(* IEC 61131-3 sources: SmartHomeNew/ (part 12) *)

(* ---- PRG_Epistemic_Integrity_Governor.st ---- *)
PROGRAM PRG_Epistemic_Integrity_Governor
VAR
    L_Now_MS : UDINT;
    L_Epistemic_Valid : BOOL := TRUE;
    L_Error_Code : UDINT := 0;
    L_Error_Text : STRING(160) := '';
END_VAR

L_Now_MS := GVL_STATUS.G_System_Time_MS;
L_Epistemic_Valid := TRUE;
L_Error_Code := 0;
L_Error_Text := '';

// Fail-safe defaults.
GVL_EPISTEMIC_INTEGRITY_FABRIC.Epistemic_Integrity_Valid := FALSE;
GVL_EPISTEMIC_INTEGRITY_FABRIC.Epistemic_Integrity_Granted := FALSE;
GVL_EPISTEMIC_INTEGRITY_FABRIC.Epistemic_Integrity_Quarantine_Active := TRUE;

GVL_EPISTEMIC_INTEGRITY_FABRIC.Physical_Reality_Model_Coherent := FALSE;
GVL_EPISTEMIC_INTEGRITY_FABRIC.Sensor_Truth_Consensus_Valid := FALSE;
GVL_EPISTEMIC_INTEGRITY_FABRIC.Telemetry_Reality_Alignment_Stable := FALSE;
GVL_EPISTEMIC_INTEGRITY_FABRIC.Distributed_Reality_Model_Consistent := FALSE;
GVL_EPISTEMIC_INTEGRITY_FABRIC.Causal_Model_Physically_Valid := FALSE;

// Forensic evidence required.
IF NOT GVL_FORENSIC_EVIDENCE_FABRIC.Forensic_Evidence_Granted THEN
    L_Epistemic_Valid := FALSE;
    L_Error_Code := 44000;
    L_Error_Text := 'Forensic evidence authority not granted';
END_IF;

// Epistemic split-brain detectors.
IF GVL_EPISTEMIC_INTEGRITY_FABRIC.Physically_False_Consensus_Detected THEN
    L_Epistemic_Valid := FALSE;
    L_Error_Code := 44001;
    L_Error_Text := 'Physically false consensus detected';
END_IF;

IF GVL_EPISTEMIC_INTEGRITY_FABRIC.Telemetry_Corruption_Coherent_Detected THEN
    L_Epistemic_Valid := FALSE;
    L_Error_Code := 44002;
    L_Error_Text := 'Telemetry corruption coherence detected';
END_IF;

IF GVL_EPISTEMIC_INTEGRITY_FABRIC.Historical_Reality_Divergence_Detected THEN
    L_Epistemic_Valid := FALSE;
    L_Error_Code := 44003;
    L_Error_Text := 'Historical reality divergence detected';
END_IF;

IF GVL_EPISTEMIC_INTEGRITY_FABRIC.Sensor_Trust_Erosion_Detected THEN
    L_Epistemic_Valid := FALSE;
    L_Error_Code := 44004;
    L_Error_Text := 'Sensor trust erosion detected';
END_IF;

IF GVL_EPISTEMIC_INTEGRITY_FABRIC.Causal_Model_Poisoning_Detected THEN
    L_Epistemic_Valid := FALSE;
    L_Error_Code := 44005;
    L_Error_Text := 'Causal model poisoning detected';
END_IF;

IF GVL_EPISTEMIC_INTEGRITY_FABRIC.LongTerm_Epistemic_Drift_Detected THEN
    L_Epistemic_Valid := FALSE;
    L_Error_Code := 44006;
    L_Error_Text := 'Long-term epistemic drift detected';
END_IF;

// Physical reality anchoring validation.
IF L_Epistemic_Valid
AND NOT GVL_EPISTEMIC_INTEGRITY_FABRIC.Historical_Reality_Anchoring_Valid THEN
    L_Epistemic_Valid := FALSE;
    L_Error_Code := 44010;
    L_Error_Text := 'Historical reality anchoring invalid';
END_IF;

IF L_Epistemic_Valid
AND NOT GVL_EPISTEMIC_INTEGRITY_FABRIC.Physical_Truth_Lineage_Coherent THEN
    L_Epistemic_Valid := FALSE;
    L_Error_Code := 44011;
    L_Error_Text := 'Physical truth lineage coherence invalid';
END_IF;

IF L_Epistemic_Valid
AND NOT GVL_EPISTEMIC_INTEGRITY_FABRIC.Reality_Model_Drift_Bounded THEN
    L_Epistemic_Valid := FALSE;
    L_Error_Code := 44012;
    L_Error_Text := 'Reality model drift bounds invalid';
END_IF;

IF L_Epistemic_Valid
AND NOT GVL_EPISTEMIC_INTEGRITY_FABRIC.Semantic_To_Physical_Causality_Valid THEN
    L_Epistemic_Valid := FALSE;
    L_Error_Code := 44013;
    L_Error_Text := 'Semantic-to-physical causality invalid';
END_IF;

IF L_Epistemic_Valid THEN
    GVL_EPISTEMIC_INTEGRITY_FABRIC.Epistemic_Integrity_Valid := TRUE;
    GVL_EPISTEMIC_INTEGRITY_FABRIC.Epistemic_Integrity_Granted := TRUE;
    GVL_EPISTEMIC_INTEGRITY_FABRIC.Epistemic_Integrity_Quarantine_Active := FALSE;

    GVL_EPISTEMIC_INTEGRITY_FABRIC.Physical_Reality_Model_Coherent := TRUE;
    GVL_EPISTEMIC_INTEGRITY_FABRIC.Sensor_Truth_Consensus_Valid := TRUE;
    GVL_EPISTEMIC_INTEGRITY_FABRIC.Telemetry_Reality_Alignment_Stable := TRUE;
    GVL_EPISTEMIC_INTEGRITY_FABRIC.Distributed_Reality_Model_Consistent := TRUE;
    GVL_EPISTEMIC_INTEGRITY_FABRIC.Causal_Model_Physically_Valid := TRUE;

    GVL_EPISTEMIC_INTEGRITY_FABRIC.Epistemic_Integrity_Epoch :=
        GVL_FORENSIC_EVIDENCE_FABRIC.Forensic_Evidence_Epoch;

    GVL_EPISTEMIC_INTEGRITY_FABRIC.Epistemic_Integrity_Epoch_Coherent := TRUE;

    GVL_EPISTEMIC_INTEGRITY_FABRIC.Epistemic_Integrity_Last_Update_MS :=
        L_Now_MS;

    GVL_EPISTEMIC_INTEGRITY_FABRIC.Epistemic_Integrity_Lease_Expired := FALSE;

    GVL_EPISTEMIC_INTEGRITY_FABRIC.Epistemic_Integrity_Last_Error_Code := 0;
    GVL_EPISTEMIC_INTEGRITY_FABRIC.Epistemic_Integrity_Last_Error_Text := '';
ELSE
    GVL_EPISTEMIC_INTEGRITY_FABRIC.Epistemic_Integrity_Valid := FALSE;
    GVL_EPISTEMIC_INTEGRITY_FABRIC.Epistemic_Integrity_Granted := FALSE;
    GVL_EPISTEMIC_INTEGRITY_FABRIC.Epistemic_Integrity_Quarantine_Active := TRUE;

    GVL_EPISTEMIC_INTEGRITY_FABRIC.Epistemic_Integrity_Lease_Expired := TRUE;

    GVL_EPISTEMIC_INTEGRITY_FABRIC.Epistemic_Integrity_Last_Error_Code :=
        L_Error_Code;

    GVL_EPISTEMIC_INTEGRITY_FABRIC.Epistemic_Integrity_Last_Error_Text :=
        L_Error_Text;

    GVL_EPISTEMIC_INTEGRITY_FABRIC.Epistemic_Integrity_Invalidation_Count :=
        GVL_EPISTEMIC_INTEGRITY_FABRIC.Epistemic_Integrity_Invalidation_Count + 1;
END_IF;

END_PROGRAM

(* ---- PRG_Execution_Progress_Causality_Governor.st ---- *)
PROGRAM PRG_Execution_Progress_Causality_Governor
IF GVL_PHYSICAL_DEADLOCK_RESOLUTION_FABRIC.Physical_Deadlock_Resolution_Granted
AND NOT GVL_EXECUTION_PROGRESS_CAUSALITY_FABRIC.Distributed_Execution_Stall_Detected
AND NOT GVL_EXECUTION_PROGRESS_CAUSALITY_FABRIC.Execution_Progress_Divergence_Detected
AND NOT GVL_EXECUTION_PROGRESS_CAUSALITY_FABRIC.Recovery_Progress_Oscillation_Detected THEN

    GVL_EXECUTION_PROGRESS_CAUSALITY_FABRIC.Execution_Progress_Causality_Valid := TRUE;
    GVL_EXECUTION_PROGRESS_CAUSALITY_FABRIC.Execution_Progress_Causality_Granted := TRUE;
    GVL_EXECUTION_PROGRESS_CAUSALITY_FABRIC.Progress_Causality_Grounded := TRUE;
    GVL_EXECUTION_PROGRESS_CAUSALITY_FABRIC.Deterministic_Execution_Continuation_Valid := TRUE;
END_IF;
END_PROGRAM

(* ---- PRG_Explainability.st ---- *)
PROGRAM PRG_Explainability
VAR
    L_Mode : E_Safety_Mode;
    L_Recovery : E_Recovery_Phase;
END_VAR

L_Mode := GVL_SAFETY_SHUTDOWN.G_Safety_Mode;
L_Recovery := GVL_SAFETY_RECOVERY.G_Recovery_Phase;

GVL_EXPLAINABILITY.G_Last_Safety_Mode := L_Mode;
GVL_EXPLAINABILITY.G_Last_Recovery_Phase := L_Recovery;
GVL_EXPLAINABILITY.G_Last_Update_MS := GVL_TIME_SERVICE.G_Now_MS;

// Global reason
CASE L_Mode OF
    FIRE:
        GVL_EXPLAINABILITY.G_Last_Global_Reason_Code := REASON_FIRE;
        GVL_EXPLAINABILITY.G_Last_Global_Reason_Text := 'Fire safety mode active';
    GAS:
        GVL_EXPLAINABILITY.G_Last_Global_Reason_Code := REASON_GAS;
        GVL_EXPLAINABILITY.G_Last_Global_Reason_Text := 'Gas safety mode active';
    WATER_LEAK:
        GVL_EXPLAINABILITY.G_Last_Global_Reason_Code := REASON_WATER_LEAK;
        GVL_EXPLAINABILITY.G_Last_Global_Reason_Text := 'Water leak detected';
    GLOBAL_STOP:
        GVL_EXPLAINABILITY.G_Last_Global_Reason_Code := REASON_GLOBAL_STOP;
        GVL_EXPLAINABILITY.G_Last_Global_Reason_Text := 'Global stop active';
    EVACUATION:
        GVL_EXPLAINABILITY.G_Last_Global_Reason_Code := REASON_EVACUATION;
        GVL_EXPLAINABILITY.G_Last_Global_Reason_Text := 'Evacuation mode active';
    NORMAL:
        IF GVL_SAFETY_RECOVERY.G_Recovery_Active THEN
            GVL_EXPLAINABILITY.G_Last_Global_Reason_Code := REASON_RECOVERY_ACTIVE;
            GVL_EXPLAINABILITY.G_Last_Global_Reason_Text := 'System in recovery phase';
        ELSE
            GVL_EXPLAINABILITY.G_Last_Global_Reason_Code := REASON_NONE;
            GVL_EXPLAINABILITY.G_Last_Global_Reason_Text := 'System in normal operation';
        END_IF;
END_CASE;

// Domain explanations
IF GVL_COMMAND_SHADOW.G_Heating_Block THEN
    GVL_EXPLAINABILITY.G_Heating_Why_Blocked := 'Heating blocked by command arbitration (safety or recovery)';
ELSE
    GVL_EXPLAINABILITY.G_Heating_Why_Blocked := '';
END_IF;

IF GVL_COMMAND_SHADOW.G_Vent_Stop THEN
    GVL_EXPLAINABILITY.G_Vent_Why_Stopped := 'Ventilation stopped by command arbitration';
ELSE
    GVL_EXPLAINABILITY.G_Vent_Why_Stopped := '';
END_IF;

IF GVL_COMMAND_SHADOW.G_Close_Valve_35 OR GVL_COMMAND_SHADOW.G_Close_Valve_36 THEN
    GVL_EXPLAINABILITY.G_Water_Why_Closed := 'Water valves closed by safety command';
ELSE
    GVL_EXPLAINABILITY.G_Water_Why_Closed := '';
END_IF;

IF GVL_COMMAND_SHADOW.G_Lock_1_Open OR GVL_COMMAND_SHADOW.G_Lock_2_Open THEN
    GVL_EXPLAINABILITY.G_Access_Why_Opened := 'Access opened due to evacuation or command override';
ELSE
    GVL_EXPLAINABILITY.G_Access_Why_Opened := '';
END_IF;

// >>> BULK_SYNC_ANCHOR: PRG_Explainability <<<

(* ---- PRG_File_Archive_HMI_Applicator.st ---- *)
PROGRAM PRG_File_Archive_HMI_Applicator
// ==============================================================================
// FILE ARCHIVE HMI APPLICATOR — validates HMI intent and updates archive runtime.
// ==============================================================================
// HMI is not allowed to write files or physical outputs directly. This program
// only transfers validated one-shot requests/configuration into GVL_FILE_ARCHIVE,
// where PRG_File_Archive_Manager consumes them and publishes deterministic status.
// ==============================================================================
VAR
    L_Any_Write_Request : BOOL;
END_VAR

L_Any_Write_Request :=
    GVL_FILE_ARCHIVE_HMI.G_Write_Event_CSV_Req
    OR GVL_FILE_ARCHIVE_HMI.G_Write_Trend_CSV_Req
    OR GVL_FILE_ARCHIVE_HMI.G_Write_BlackBox_CSV_Req
    OR GVL_FILE_ARCHIVE_HMI.G_Write_Config_Backup_Req;

IF GVL_FILE_ARCHIVE_HMI.G_Set_Archive_Config_Req THEN
    IF GVL_FILE_ARCHIVE_HMI.G_File_Archive_Target_Code <= 3 THEN
        GVL_FILE_ARCHIVE.G_Archive_Interface_Enabled := GVL_FILE_ARCHIVE_HMI.G_Archive_Interface_Enabled;
        GVL_FILE_ARCHIVE.G_CSV_Write_Enabled := GVL_FILE_ARCHIVE_HMI.G_CSV_Write_Enabled;
        GVL_FILE_ARCHIVE.G_File_Archive_Target_Code := GVL_FILE_ARCHIVE_HMI.G_File_Archive_Target_Code;

        GVL_FILE_ARCHIVE_HMI.G_Last_Error := FALSE;
        GVL_FILE_ARCHIVE_HMI.G_Last_Error_Code := 0;
        GVL_FILE_ARCHIVE_HMI.G_Last_Status_Text := 'Archive configuration applied';
    ELSE
        GVL_FILE_ARCHIVE_HMI.G_Last_Error := TRUE;
        GVL_FILE_ARCHIVE_HMI.G_Last_Error_Code := 16#A101;
        GVL_FILE_ARCHIVE_HMI.G_Last_Status_Text := 'Archive configuration rejected: invalid target';
    END_IF;

    GVL_FILE_ARCHIVE_HMI.G_Last_Update_MS := GVL_TIME_SERVICE.G_Now_MS;
    GVL_FILE_ARCHIVE_HMI.G_Set_Archive_Config_Req := FALSE;
END_IF;

IF L_Any_Write_Request THEN
    IF NOT GVL_FILE_ARCHIVE.G_Archive_Interface_Enabled THEN
        GVL_FILE_ARCHIVE_HMI.G_Last_Error := TRUE;
        GVL_FILE_ARCHIVE_HMI.G_Last_Error_Code := 16#A102;
        GVL_FILE_ARCHIVE_HMI.G_Last_Status_Text := 'Archive write rejected: interface disabled';
    ELSIF NOT GVL_FILE_ARCHIVE.G_CSV_Write_Enabled THEN
        GVL_FILE_ARCHIVE_HMI.G_Last_Error := TRUE;
        GVL_FILE_ARCHIVE_HMI.G_Last_Error_Code := 16#A103;
        GVL_FILE_ARCHIVE_HMI.G_Last_Status_Text := 'Archive write rejected: CSV disabled';
    ELSE
        GVL_FILE_ARCHIVE.G_Write_Event_CSV_Request :=
            GVL_FILE_ARCHIVE.G_Write_Event_CSV_Request OR GVL_FILE_ARCHIVE_HMI.G_Write_Event_CSV_Req;
        GVL_FILE_ARCHIVE.G_Write_Trend_CSV_Request :=
            GVL_FILE_ARCHIVE.G_Write_Trend_CSV_Request OR GVL_FILE_ARCHIVE_HMI.G_Write_Trend_CSV_Req;
        GVL_FILE_ARCHIVE.G_Write_BlackBox_CSV_Request :=
            GVL_FILE_ARCHIVE.G_Write_BlackBox_CSV_Request OR GVL_FILE_ARCHIVE_HMI.G_Write_BlackBox_CSV_Req;
        GVL_FILE_ARCHIVE.G_Write_Config_Backup_Request :=
            GVL_FILE_ARCHIVE.G_Write_Config_Backup_Request OR GVL_FILE_ARCHIVE_HMI.G_Write_Config_Backup_Req;

        GVL_FILE_ARCHIVE_HMI.G_Last_Error := FALSE;
        GVL_FILE_ARCHIVE_HMI.G_Last_Error_Code := 0;
        GVL_FILE_ARCHIVE_HMI.G_Last_Status_Text := 'Archive write request accepted';
    END_IF;

    GVL_FILE_ARCHIVE_HMI.G_Last_Update_MS := GVL_TIME_SERVICE.G_Now_MS;

    // HMI requests are one-shot. Runtime requests are consumed by archive manager.
    GVL_FILE_ARCHIVE_HMI.G_Write_Event_CSV_Req := FALSE;
    GVL_FILE_ARCHIVE_HMI.G_Write_Trend_CSV_Req := FALSE;
    GVL_FILE_ARCHIVE_HMI.G_Write_BlackBox_CSV_Req := FALSE;
    GVL_FILE_ARCHIVE_HMI.G_Write_Config_Backup_Req := FALSE;
END_IF;

// >>> BULK_SYNC_ANCHOR: PRG_File_Archive_HMI_Applicator <<<
END_PROGRAM

(* ---- PRG_File_Archive_Manager.st ---- *)
PROGRAM PRG_File_Archive_Manager
// ==============================================================================
// FILE ARCHIVE MANAGER — deterministic runtime surface for future CSV/file export.
// ==============================================================================
// No direct file, USB or gateway write is implemented here. This program only
// consumes one-shot archive requests, validates the configured target surface and
// publishes a deterministic status/error until concrete CODESYS file libraries
// and port-specific paths are selected.
// ==============================================================================
VAR
    L_Request_Active : BOOL;
    L_Target_Available : BOOL;
END_VAR

L_Request_Active :=
    GVL_FILE_ARCHIVE.G_Write_Event_CSV_Request
    OR GVL_FILE_ARCHIVE.G_Write_Trend_CSV_Request
    OR GVL_FILE_ARCHIVE.G_Write_BlackBox_CSV_Request
    OR GVL_FILE_ARCHIVE.G_Write_Config_Backup_Request;

L_Target_Available := FALSE;
CASE GVL_FILE_ARCHIVE.G_File_Archive_Target_Code OF
    1:
        L_Target_Available := GVL_FILE_ARCHIVE.G_PLC_File_Target_Available;
    2:
        L_Target_Available := GVL_FILE_ARCHIVE.G_USB_Target_Available;
    3:
        L_Target_Available := GVL_FILE_ARCHIVE.G_Gateway_Target_Available;
ELSE
    L_Target_Available := FALSE;
END_CASE;

IF L_Request_Active THEN
    GVL_FILE_ARCHIVE.G_Write_Busy := FALSE;
    GVL_FILE_ARCHIVE.G_Write_Done := FALSE;
    GVL_FILE_ARCHIVE.G_Write_Error := FALSE;
    GVL_FILE_ARCHIVE.G_Last_Error_Code := 0;
    GVL_FILE_ARCHIVE.G_Last_Status_Text := '';
    GVL_FILE_ARCHIVE.G_Last_Write_MS := GVL_TIME_SERVICE.G_Now_MS;

    IF NOT GVL_FILE_ARCHIVE.G_Archive_Interface_Enabled THEN
        GVL_FILE_ARCHIVE.G_Write_Error := TRUE;
        GVL_FILE_ARCHIVE.G_Last_Error_Code := 16#A001;
        GVL_FILE_ARCHIVE.G_Last_Status_Text := 'Archive interface disabled';
    ELSIF NOT GVL_FILE_ARCHIVE.G_CSV_Write_Enabled THEN
        GVL_FILE_ARCHIVE.G_Write_Error := TRUE;
        GVL_FILE_ARCHIVE.G_Last_Error_Code := 16#A002;
        GVL_FILE_ARCHIVE.G_Last_Status_Text := 'CSV archive disabled';
    ELSIF GVL_FILE_ARCHIVE.G_File_Archive_Target_Code = 0 THEN
        GVL_FILE_ARCHIVE.G_Write_Error := TRUE;
        GVL_FILE_ARCHIVE.G_Last_Error_Code := 16#A003;
        GVL_FILE_ARCHIVE.G_Last_Status_Text := 'No archive target selected';
    ELSIF NOT L_Target_Available THEN
        GVL_FILE_ARCHIVE.G_Write_Error := TRUE;
        GVL_FILE_ARCHIVE.G_Last_Error_Code := 16#A004;
        GVL_FILE_ARCHIVE.G_Last_Status_Text := 'Selected archive target unavailable';
    ELSE
        GVL_FILE_ARCHIVE.G_Write_Error := TRUE;
        GVL_FILE_ARCHIVE.G_Last_Error_Code := 16#A005;
        GVL_FILE_ARCHIVE.G_Last_Status_Text := 'Archive backend not connected';
    END_IF;

    // One-shot requests are consumed regardless of the result so HMI/gateway
    // callers receive a stable status instead of repeatedly retriggering.
    GVL_FILE_ARCHIVE.G_Write_Event_CSV_Request := FALSE;
    GVL_FILE_ARCHIVE.G_Write_Trend_CSV_Request := FALSE;
    GVL_FILE_ARCHIVE.G_Write_BlackBox_CSV_Request := FALSE;
    GVL_FILE_ARCHIVE.G_Write_Config_Backup_Request := FALSE;
END_IF;

// >>> BULK_SYNC_ANCHOR: PRG_File_Archive_Manager <<<
END_PROGRAM

(* ---- PRG_Governance_Observer_Consensus_Governor.st ---- *)
PROGRAM PRG_Governance_Observer_Consensus_Governor
VAR
    L_Now_MS : UDINT;
    L_Consensus_Valid : BOOL := TRUE;
    L_Error_Code : UDINT := 0;
    L_Error_Text : STRING(160) := '';
END_VAR

L_Now_MS := GVL_STATUS.G_System_Time_MS;
L_Consensus_Valid := TRUE;
L_Error_Code := 0;
L_Error_Text := '';

// Fail-safe defaults.
GVL_GOVERNANCE_OBSERVER_CONSENSUS_FABRIC.Governance_Observer_Consensus_Valid := FALSE;
GVL_GOVERNANCE_OBSERVER_CONSENSUS_FABRIC.Governance_Observer_Consensus_Granted := FALSE;
GVL_GOVERNANCE_OBSERVER_CONSENSUS_FABRIC.Governance_Observer_Consensus_Quarantine_Active := TRUE;

GVL_GOVERNANCE_OBSERVER_CONSENSUS_FABRIC.Distributed_Governance_Projection_Consistent := FALSE;
GVL_GOVERNANCE_OBSERVER_CONSENSUS_FABRIC.Observer_Semantic_Consensus_Valid := FALSE;
GVL_GOVERNANCE_OBSERVER_CONSENSUS_FABRIC.CrossNode_Authority_Interpretation_Aligned := FALSE;
GVL_GOVERNANCE_OBSERVER_CONSENSUS_FABRIC.Governance_Reality_Canonical := FALSE;
GVL_GOVERNANCE_OBSERVER_CONSENSUS_FABRIC.Observer_Projection_Lineage_Coherent := FALSE;

// Semantic epoch invariance required.
IF NOT GVL_SEMANTIC_EPOCH_INVARIANCE_FABRIC.Semantic_Epoch_Invariance_Granted THEN
    L_Consensus_Valid := FALSE;
    L_Error_Code := 50000;
    L_Error_Text := 'Semantic epoch invariance not granted';
END_IF;

// Governance observer split-brain detectors.
IF GVL_GOVERNANCE_OBSERVER_CONSENSUS_FABRIC.Observer_Governance_Divergence_Detected THEN
    L_Consensus_Valid := FALSE;
    L_Error_Code := 50001;
    L_Error_Text := 'Observer governance divergence detected';
END_IF;

IF GVL_GOVERNANCE_OBSERVER_CONSENSUS_FABRIC.CrossNode_Authority_Interpretation_Fork THEN
    L_Consensus_Valid := FALSE;
    L_Error_Code := 50002;
    L_Error_Text := 'Cross-node authority interpretation fork detected';
END_IF;

IF GVL_GOVERNANCE_OBSERVER_CONSENSUS_FABRIC.Semantic_Projection_Mismatch_Detected THEN
    L_Consensus_Valid := FALSE;
    L_Error_Code := 50003;
    L_Error_Text := 'Semantic projection mismatch detected';
END_IF;

IF GVL_GOVERNANCE_OBSERVER_CONSENSUS_FABRIC.Canonical_Governance_Reality_Lost THEN
    L_Consensus_Valid := FALSE;
    L_Error_Code := 50004;
    L_Error_Text := 'Canonical governance reality lost';
END_IF;

IF GVL_GOVERNANCE_OBSERVER_CONSENSUS_FABRIC.Observer_Projection_Lineage_Drift_Detected THEN
    L_Consensus_Valid := FALSE;
    L_Error_Code := 50005;
    L_Error_Text := 'Observer projection lineage drift detected';
END_IF;

IF GVL_GOVERNANCE_OBSERVER_CONSENSUS_FABRIC.Distributed_Governance_Reality_Fork_Detected THEN
    L_Consensus_Valid := FALSE;
    L_Error_Code := 50006;
    L_Error_Text := 'Distributed governance reality fork detected';
END_IF;

// Observer consensus validation.
IF L_Consensus_Valid
AND NOT GVL_GOVERNANCE_OBSERVER_CONSENSUS_FABRIC.Canonical_Projection_Vector_Stable THEN
    L_Consensus_Valid := FALSE;
    L_Error_Code := 50010;
    L_Error_Text := 'Canonical projection vector invalid';
END_IF;

IF L_Consensus_Valid
AND NOT GVL_GOVERNANCE_OBSERVER_CONSENSUS_FABRIC.Distributed_Interpretation_Equivalence_Valid THEN
    L_Consensus_Valid := FALSE;
    L_Error_Code := 50011;
    L_Error_Text := 'Distributed interpretation equivalence invalid';
END_IF;

IF L_Consensus_Valid
AND NOT GVL_GOVERNANCE_OBSERVER_CONSENSUS_FABRIC.Governance_Projection_Causality_Grounded THEN
    L_Consensus_Valid := FALSE;
    L_Error_Code := 50012;
    L_Error_Text := 'Governance projection causality invalid';
END_IF;

IF L_Consensus_Valid
AND NOT GVL_GOVERNANCE_OBSERVER_CONSENSUS_FABRIC.Observer_Timeline_Consensus_Monotonic THEN
    L_Consensus_Valid := FALSE;
    L_Error_Code := 50013;
    L_Error_Text := 'Observer timeline consensus monotonicity invalid';
END_IF;

IF L_Consensus_Valid THEN
    GVL_GOVERNANCE_OBSERVER_CONSENSUS_FABRIC.Governance_Observer_Consensus_Valid := TRUE;
    GVL_GOVERNANCE_OBSERVER_CONSENSUS_FABRIC.Governance_Observer_Consensus_Granted := TRUE;
    GVL_GOVERNANCE_OBSERVER_CONSENSUS_FABRIC.Governance_Observer_Consensus_Quarantine_Active := FALSE;

    GVL_GOVERNANCE_OBSERVER_CONSENSUS_FABRIC.Distributed_Governance_Projection_Consistent := TRUE;
    GVL_GOVERNANCE_OBSERVER_CONSENSUS_FABRIC.Observer_Semantic_Consensus_Valid := TRUE;
    GVL_GOVERNANCE_OBSERVER_CONSENSUS_FABRIC.CrossNode_Authority_Interpretation_Aligned := TRUE;
    GVL_GOVERNANCE_OBSERVER_CONSENSUS_FABRIC.Governance_Reality_Canonical := TRUE;
    GVL_GOVERNANCE_OBSERVER_CONSENSUS_FABRIC.Observer_Projection_Lineage_Coherent := TRUE;

    GVL_GOVERNANCE_OBSERVER_CONSENSUS_FABRIC.Governance_Observer_Consensus_Epoch :=
        GVL_SEMANTIC_EPOCH_INVARIANCE_FABRIC.Semantic_Epoch_Invariance_Epoch;

    GVL_GOVERNANCE_OBSERVER_CONSENSUS_FABRIC.Governance_Observer_Consensus_Epoch_Coherent := TRUE;

    GVL_GOVERNANCE_OBSERVER_CONSENSUS_FABRIC.Governance_Observer_Consensus_Last_Update_MS :=
        L_Now_MS;

    GVL_GOVERNANCE_OBSERVER_CONSENSUS_FABRIC.Governance_Observer_Consensus_Lease_Expired := FALSE;

    GVL_GOVERNANCE_OBSERVER_CONSENSUS_FABRIC.Governance_Observer_Consensus_Last_Error_Code := 0;
    GVL_GOVERNANCE_OBSERVER_CONSENSUS_FABRIC.Governance_Observer_Consensus_Last_Error_Text := '';
ELSE
    GVL_GOVERNANCE_OBSERVER_CONSENSUS_FABRIC.Governance_Observer_Consensus_Valid := FALSE;
    GVL_GOVERNANCE_OBSERVER_CONSENSUS_FABRIC.Governance_Observer_Consensus_Granted := FALSE;
    GVL_GOVERNANCE_OBSERVER_CONSENSUS_FABRIC.Governance_Observer_Consensus_Quarantine_Active := TRUE;

    GVL_GOVERNANCE_OBSERVER_CONSENSUS_FABRIC.Governance_Observer_Consensus_Lease_Expired := TRUE;

    GVL_GOVERNANCE_OBSERVER_CONSENSUS_FABRIC.Governance_Observer_Consensus_Last_Error_Code :=
        L_Error_Code;

    GVL_GOVERNANCE_OBSERVER_CONSENSUS_FABRIC.Governance_Observer_Consensus_Last_Error_Text :=
        L_Error_Text;

    GVL_GOVERNANCE_OBSERVER_CONSENSUS_FABRIC.Governance_Observer_Consensus_Invalidation_Count :=
        GVL_GOVERNANCE_OBSERVER_CONSENSUS_FABRIC.Governance_Observer_Consensus_Invalidation_Count + 1;
END_IF;

END_PROGRAM

(* ---- PRG_Governance_Publication_Binding_Governor.st ---- *)
PROGRAM PRG_Governance_Publication_Binding_Governor
VAR
    L_Now_MS : UDINT;
    L_Valid : BOOL := TRUE;
    L_Error_Code : UDINT := 0;
    L_Error_Text : STRING(160) := '';
END_VAR

L_Now_MS := GVL_STATUS.G_System_Time_MS;
L_Valid := TRUE;
L_Error_Code := 0;
L_Error_Text := '';

// Fail-safe defaults.
GVL_GOVERNANCE_PUBLICATION_BINDING_FABRIC.Governance_Publication_Binding_Valid := FALSE;
GVL_GOVERNANCE_PUBLICATION_BINDING_FABRIC.Governance_Publication_Binding_Granted := FALSE;
GVL_GOVERNANCE_PUBLICATION_BINDING_FABRIC.Governance_Publication_Binding_Quarantine_Active := TRUE;

GVL_GOVERNANCE_PUBLICATION_BINDING_FABRIC.Observability_Publication_Causality_Valid := FALSE;
GVL_GOVERNANCE_PUBLICATION_BINDING_FABRIC.Upstream_Governance_Lease_Fresh := FALSE;
GVL_GOVERNANCE_PUBLICATION_BINDING_FABRIC.Governance_Publication_Epoch_Coherent := FALSE;
GVL_GOVERNANCE_PUBLICATION_BINDING_FABRIC.Publication_Quarantine_Propagation_Valid := FALSE;
GVL_GOVERNANCE_PUBLICATION_BINDING_FABRIC.Canonical_Observability_Reality_Consistent := FALSE;

// Governance liveness integrity required.
IF NOT GVL_GOVERNANCE_LIVENESS_INTEGRITY_FABRIC.Governance_Liveness_Integrity_Granted THEN
    L_Valid := FALSE;
    L_Error_Code := 55000;
    L_Error_Text := 'Governance liveness integrity not granted';
END_IF;

// Publication binding detectors.
IF GVL_GOVERNANCE_PUBLICATION_BINDING_FABRIC.Stale_Valid_Publication_Detected THEN
    L_Valid := FALSE;
    L_Error_Code := 55001;
    L_Error_Text := 'Stale valid publication detected';
END_IF;

IF GVL_GOVERNANCE_PUBLICATION_BINDING_FABRIC.LeaseExpired_Governance_Published_As_Healthy THEN
    L_Valid := FALSE;
    L_Error_Code := 55002;
    L_Error_Text := 'Lease-expired governance published as healthy';
END_IF;

IF GVL_GOVERNANCE_PUBLICATION_BINDING_FABRIC.Quarantine_State_Publication_Bypass THEN
    L_Valid := FALSE;
    L_Error_Code := 55003;
    L_Error_Text := 'Quarantine state publication bypass';
END_IF;

IF GVL_GOVERNANCE_PUBLICATION_BINDING_FABRIC.Governance_Invalidation_Hidden_From_Observability THEN
    L_Valid := FALSE;
    L_Error_Code := 55004;
    L_Error_Text := 'Governance invalidation hidden from observability';
END_IF;

IF GVL_GOVERNANCE_PUBLICATION_BINDING_FABRIC.Distributed_Publication_State_Fork_Detected THEN
    L_Valid := FALSE;
    L_Error_Code := 55005;
    L_Error_Text := 'Distributed publication state fork detected';
END_IF;

IF GVL_GOVERNANCE_PUBLICATION_BINDING_FABRIC.Historical_Invalidation_Causality_Lost THEN
    L_Valid := FALSE;
    L_Error_Code := 55006;
    L_Error_Text := 'Historical invalidation causality lost';
END_IF;

// Publication validation.
IF L_Valid
AND NOT GVL_GOVERNANCE_PUBLICATION_BINDING_FABRIC.Diagnostics_Publication_Consistency_Valid THEN
    L_Valid := FALSE;
    L_Error_Code := 55010;
    L_Error_Text := 'Diagnostics publication consistency invalid';
END_IF;

IF L_Valid
AND NOT GVL_GOVERNANCE_PUBLICATION_BINDING_FABRIC.HMI_Publication_State_Aligned THEN
    L_Valid := FALSE;
    L_Error_Code := 55011;
    L_Error_Text := 'HMI publication state alignment invalid';
END_IF;

IF L_Valid
AND NOT GVL_GOVERNANCE_PUBLICATION_BINDING_FABRIC.Blackbox_Invalidation_Lineage_Valid THEN
    L_Valid := FALSE;
    L_Error_Code := 55012;
    L_Error_Text := 'Blackbox invalidation lineage invalid';
END_IF;

IF L_Valid
AND NOT GVL_GOVERNANCE_PUBLICATION_BINDING_FABRIC.Distributed_Publication_Consensus_Valid THEN
    L_Valid := FALSE;
    L_Error_Code := 55013;
    L_Error_Text := 'Distributed publication consensus invalid';
END_IF;

IF L_Valid THEN
    GVL_GOVERNANCE_PUBLICATION_BINDING_FABRIC.Governance_Publication_Binding_Valid := TRUE;
    GVL_GOVERNANCE_PUBLICATION_BINDING_FABRIC.Governance_Publication_Binding_Granted := TRUE;
    GVL_GOVERNANCE_PUBLICATION_BINDING_FABRIC.Governance_Publication_Binding_Quarantine_Active := FALSE;

    GVL_GOVERNANCE_PUBLICATION_BINDING_FABRIC.Observability_Publication_Causality_Valid := TRUE;
    GVL_GOVERNANCE_PUBLICATION_BINDING_FABRIC.Upstream_Governance_Lease_Fresh := TRUE;
    GVL_GOVERNANCE_PUBLICATION_BINDING_FABRIC.Governance_Publication_Epoch_Coherent := TRUE;
    GVL_GOVERNANCE_PUBLICATION_BINDING_FABRIC.Publication_Quarantine_Propagation_Valid := TRUE;
    GVL_GOVERNANCE_PUBLICATION_BINDING_FABRIC.Canonical_Observability_Reality_Consistent := TRUE;

    GVL_GOVERNANCE_PUBLICATION_BINDING_FABRIC.Governance_Publication_Binding_Epoch :=
        GVL_GOVERNANCE_LIVENESS_INTEGRITY_FABRIC.Governance_Liveness_Integrity_Epoch;

    GVL_GOVERNANCE_PUBLICATION_BINDING_FABRIC.Governance_Publication_Binding_Epoch_Coherent_Runtime := TRUE;

    GVL_GOVERNANCE_PUBLICATION_BINDING_FABRIC.Governance_Publication_Binding_Last_Update_MS :=
        L_Now_MS;

    GVL_GOVERNANCE_PUBLICATION_BINDING_FABRIC.Governance_Publication_Binding_Lease_Expired := FALSE;

    GVL_GOVERNANCE_PUBLICATION_BINDING_FABRIC.Governance_Publication_Binding_Last_Error_Code := 0;
    GVL_GOVERNANCE_PUBLICATION_BINDING_FABRIC.Governance_Publication_Binding_Last_Error_Text := '';
ELSE
    GVL_GOVERNANCE_PUBLICATION_BINDING_FABRIC.Governance_Publication_Binding_Valid := FALSE;
    GVL_GOVERNANCE_PUBLICATION_BINDING_FABRIC.Governance_Publication_Binding_Granted := FALSE;
    GVL_GOVERNANCE_PUBLICATION_BINDING_FABRIC.Governance_Publication_Binding_Quarantine_Active := TRUE;

    GVL_GOVERNANCE_PUBLICATION_BINDING_FABRIC.Governance_Publication_Binding_Lease_Expired := TRUE;

    GVL_GOVERNANCE_PUBLICATION_BINDING_FABRIC.Governance_Publication_Binding_Last_Error_Code :=
        L_Error_Code;

    GVL_GOVERNANCE_PUBLICATION_BINDING_FABRIC.Governance_Publication_Binding_Last_Error_Text :=
        L_Error_Text;

    GVL_GOVERNANCE_PUBLICATION_BINDING_FABRIC.Governance_Publication_Binding_Invalidation_Count :=
        GVL_GOVERNANCE_PUBLICATION_BINDING_FABRIC.Governance_Publication_Binding_Invalidation_Count + 1;
END_IF;

END_PROGRAM

(* ---- PRG_Heating.st ---- *)
PROGRAM PRG_Heating
VAR
    fbHeatingManager : FB_Heating_System_Manager;
    fbDHWManager : FB_DHW_Manager;
    fbDiagnosticsPhase : FB_Heating_Runtime_Diagnostics_Phase;
    fbObserverPhase : FB_Heating_Runtime_Observer_Phase;
    fbMetaSupervisionPublisher : FB_Heating_Runtime_Meta_Supervision_Publisher;
    fbExplainabilityPublisher : FB_Heating_Runtime_Explainability_Publisher;
    fbServiceGatingPhase : FB_Heating_Runtime_Service_Gating_Phase;
    fbStatePublicationPhase : FB_Heating_Runtime_State_Publication_Phase;
    fbOutputProjectionPhase : FB_Heating_Runtime_Output_Projection_Phase;

    L_Runtime_Context : ST_Heating_Runtime_Context;

    L_i : INT;
    L_Current_Hour : UINT;
    L_Boiler_Modulation_REAL : ARRAY[1..GVL_CONSTANTS.C_MAX_BOILERS] OF REAL;
    L_Room_Temps_Normalized : ARRAY[1..GVL_CONSTANTS.C_MAX_ZONES] OF REAL;
    L_Floor_Temps_Normalized : ARRAY[1..GVL_CONSTANTS.C_MAX_HEATING_CIRCUITS] OF REAL;
    L_Outdoor_Temp_Normalized : REAL;

    L_Heating_Emergency_Stop : BOOL;
    L_Heating_Gas_Safety_Stop : BOOL;

    L_Distributed_Execute_Allowed : BOOL;
    L_Distributed_Orchestrate_Allowed : BOOL;
    L_Distributed_Projection_Allowed : BOOL;

    L_Zone_Valves : ARRAY[1..GVL_CONSTANTS.C_MAX_HEATING_CIRCUITS] OF BOOL;
    L_Manifold_Pumps : ARRAY[1..GVL_CONSTANTS.C_MAX_MANIFOLDS] OF BOOL;
    L_Manifold_Valves : ARRAY[1..GVL_CONSTANTS.C_MAX_MANIFOLDS] OF REAL;
    L_Boiler_OT_Enable : ARRAY[1..GVL_CONSTANTS.C_MAX_BOILERS] OF BOOL;
    L_Boiler_OT_Setpoint : ARRAY[1..GVL_CONSTANTS.C_MAX_BOILERS] OF REAL;
    L_Backup_Circulation_Pump : BOOL;
    L_Electric_Heater_Enable : BOOL;
    L_Freeze_Risk_Status : BOOL;
    L_Manifold_Status : ARRAY[1..GVL_CONSTANTS.C_MAX_MANIFOLDS] OF ST_Manifold_Status;
    L_Boiler_Status : ARRAY[1..GVL_CONSTANTS.C_MAX_BOILERS] OF ST_Boiler_Status;
    L_DHW_Heating_Pump : BOOL;
    L_DHW_Circ_Pump : BOOL;
    L_DHW_Status : ST_DHW_Status;

    L_Empty_Manifold_Status : ST_Manifold_Status;
    L_Empty_Boiler_Status : ST_Boiler_Status;
    L_Empty_DHW_Status : ST_DHW_Status;
END_VAR

// Reset local output buffers at the beginning of every PRG call.
// This prevents stale publication when manager phases are skipped by governance.
FOR L_i := 1 TO GVL_CONSTANTS.C_MAX_HEATING_CIRCUITS DO
    L_Zone_Valves[L_i] := FALSE;
END_FOR;

FOR L_i := 1 TO GVL_CONSTANTS.C_MAX_MANIFOLDS DO
    L_Manifold_Pumps[L_i] := FALSE;
    L_Manifold_Valves[L_i] := 0.0;
    L_Manifold_Status[L_i] := L_Empty_Manifold_Status;
END_FOR;

FOR L_i := 1 TO GVL_CONSTANTS.C_MAX_BOILERS DO
    L_Boiler_OT_Enable[L_i] := FALSE;
    L_Boiler_OT_Setpoint[L_i] := 0.0;
    L_Boiler_Status[L_i] := L_Empty_Boiler_Status;
END_FOR;

L_Backup_Circulation_Pump := FALSE;
L_Electric_Heater_Enable := FALSE;
L_Freeze_Risk_Status := FALSE;
L_DHW_Heating_Pump := FALSE;
L_DHW_Circ_Pump := FALSE;
L_DHW_Status := L_Empty_DHW_Status;

FOR L_i := 1 TO GVL_CONSTANTS.C_MAX_BOILERS DO
    L_Boiler_Modulation_REAL[L_i] := TO_REAL(GVL_IO.AI_Boiler_Modulation[L_i]);
END_FOR;

L_Current_Hour := TO_UINT(GVL_TIME_SERVICE.G_Time_Of_Day_MS / 3600000);

L_Outdoor_Temp_Normalized := GVL_INPUT.IN_Outdoor_Temp;

FOR L_i := 1 TO GVL_CONSTANTS.C_MAX_ZONES DO
    L_Room_Temps_Normalized[L_i] := GVL_INPUT.IN_Room_Temps[L_i];
END_FOR;

FOR L_i := 1 TO GVL_CONSTANTS.C_MAX_HEATING_CIRCUITS DO
    L_Floor_Temps_Normalized[L_i] := GVL_INPUT.IN_Floor_Temps[L_i];
END_FOR;

L_Heating_Emergency_Stop := GVL_COMMAND_SHADOW.G_Heating_Emergency_Stop;
L_Heating_Gas_Safety_Stop := GVL_COMMAND_SHADOW.G_Heating_Gas_Safety_Stop OR GVL_STATE.G_Safety_Gas_Latched;

// Centralized distributed runtime governance.
// Freeze protection and gas safety semantics remain authoritative.
L_Distributed_Execute_Allowed :=
    GVL_Distributed_Execution_Gates.G_Can_Execute;

L_Distributed_Orchestrate_Allowed :=
    GVL_Distributed_Execution_Gates.G_Can_Orchestrate;

L_Distributed_Projection_Allowed :=
    GVL_Distributed_Execution_Gates.G_Can_Own_Projection;

L_Runtime_Context.Runtime_Enabled := TRUE;
L_Runtime_Context.Runtime_Ready := TRUE;
L_Runtime_Context.Runtime_Fault := FALSE;
L_Runtime_Context.Current_Phase := E_Heating_Runtime_Phase.HRP_IDLE;

L_Runtime_Context.Allow_DHW_Phase :=
    L_Distributed_Execute_Allowed;

L_Runtime_Context.Allow_Heating_Phase :=
    L_Distributed_Orchestrate_Allowed;

L_Runtime_Context.Allow_Service_Gating_Phase := TRUE;
L_Runtime_Context.Allow_State_Publication_Phase := TRUE;
L_Runtime_Context.Allow_Diagnostics_Phase := TRUE;

L_Runtime_Context.Allow_Output_Projection_Phase :=
    L_Distributed_Projection_Allowed;

L_Runtime_Context.DHW_Executed := FALSE;
L_Runtime_Context.Heating_Executed := FALSE;
L_Runtime_Context.Service_Gating_Executed := FALSE;
L_Runtime_Context.State_Publication_Executed := FALSE;
L_Runtime_Context.Diagnostics_Executed := FALSE;
L_Runtime_Context.Output_Projection_Executed := FALSE;

L_Runtime_Context.DHW_Before_Heating_Valid := TRUE;
L_Runtime_Context.State_Publication_Before_Diagnostics_Valid := TRUE;
L_Runtime_Context.Output_Projection_Last_Valid := TRUE;

L_Runtime_Context.Diagnostics_Isolation_Valid := TRUE;
L_Runtime_Context.Explainability_Isolation_Valid := TRUE;
L_Runtime_Context.Safety_Isolation_Valid := TRUE;
L_Runtime_Context.OpenTherm_Ownership_Valid := TRUE;
L_Runtime_Context.Cascade_Ownership_Valid := TRUE;

IF NOT L_Distributed_Execute_Allowed THEN
    L_Runtime_Context.Runtime_Status_Code := 20;
    L_Runtime_Context.Runtime_Status_Text :=
        'Heating runtime blocked by distributed governance';
ELSE
    L_Runtime_Context.Runtime_Status_Code := 1;
    L_Runtime_Context.Runtime_Status_Text :=
        'Heating runtime nominal';
END_IF;

L_Runtime_Context.Current_Phase := E_Heating_Runtime_Phase.HRP_IDLE;

fbObserverPhase(
    VI_Authorization_Stage := TRUE,
    VI_Finalization_Stage := FALSE,
    VI_Runtime_Context := L_Runtime_Context,
    VI_Diagnostics_Valid := TRUE
);

IF L_Distributed_Execute_Allowed THEN

    L_Runtime_Context.Current_Phase := E_Heating_Runtime_Phase.HRP_DHW;

    fbDHWManager(
        VI_System_Time_MS := GVL_STATUS.G_System_Time_MS,
        VI_Current_TOD := GVL_STATUS.G_Current_TOD,
        VI_IsActivePLC := GVL_STATUS.G_Is_Active_PLC,
        VI_Temp := GVL_STATE.G_DHW_Temp,
        VI_Pressure := GVL_STATE.G_DHW_Pressure,
        VI_Config := GVL_CONFIG.G_DHW_Config,
        VI_Current_Day_Of_Week := GVL_STATUS.G_Current_Day,
        VI_IO_Modules_Online := GVL_STATUS.G_IO_Modules_Online,
        VI_Reset_Errors := GVL_INTENT_USER.I_Reset_Errors,
        VI_Emergency_Stop := L_Heating_Emergency_Stop,
        VI_System_Mode := GVL_STATE.G_System_Mode,
        VO_Status => L_DHW_Status,
        VO_Heating_Pump => L_DHW_Heating_Pump,
        VO_Circ_Pump => L_DHW_Circ_Pump
    );

    L_Runtime_Context.DHW_Executed := TRUE;

END_IF;

IF L_Heating_Gas_Safety_Stop THEN
    L_DHW_Heating_Pump := FALSE;
    L_DHW_Status.Heating_Pump_On := FALSE;
END_IF;

IF L_Distributed_Orchestrate_Allowed THEN

    L_Runtime_Context.Current_Phase := E_Heating_Runtime_Phase.HRP_HEATING;

    fbHeatingManager(
        VI_System_Mode := GVL_STATE.G_System_Mode,
        VI_System_Time_MS := GVL_STATUS.G_System_Time_MS,
        VI_IsActivePLC := GVL_STATUS.G_Is_Active_PLC,
        VI_Outdoor_Temp := L_Outdoor_Temp_Normalized,
        VI_Config := GVL_CONFIG.G_Heating_Config,
        VI_Tariff := GVL_CONFIG.G_HMI_Tariff_Settings,
        VI_Current_Hour := L_Current_Hour,
        VI_DHW_Heating_Demand := L_DHW_Heating_Pump,
        VI_DHW_Target_Temp := GVL_CONFIG.G_DHW_Config.Target_Temp,
        VI_Emergency_Stop := L_Heating_Emergency_Stop,
        VI_Gas_Safety_Stop := L_Heating_Gas_Safety_Stop,
        VI_Boiler_Error_Status := GVL_STATE.G_Boiler_Error,
        VI_Boiler_OT_Online := GVL_STATE.G_Boiler_OT_Online,
        VI_Boiler_Modulation := L_Boiler_Modulation_REAL,
        VI_Floor_Temps := L_Floor_Temps_Normalized,
        VI_Room_Temps := L_Room_Temps_Normalized,
        VI_Manifold_Pressures := GVL_STATE.G_Manifold_Pressures,
        VI_Manifold_Currents := GVL_STATE.G_Manifold_Currents,
        VI_Manifold_Temps_Supply := GVL_STATE.G_Manifold_T_Supply,
        VI_Manifold_Temps_Return := GVL_STATE.G_Manifold_T_Return,
        VI_Boiler_Flame_Status := GVL_STATE.G_Boiler_Flame,
        VI_Zone_Configs := GVL_CONFIG.G_HMI_FloorHeating_Configs,
        VI_Rule_Actions := GVL_STATE.G_Rule_Actions,
        VI_IO_Modules_Online := GVL_STATUS.G_IO_Modules_Online,
        VI_Manifold_End_Switches := GVL_STATE.G_Manifold_End_Switches,
        VI_Valve_Test_Config := GVL_CONFIG.G_Valve_Test_Config,
        VO_Manifold_Valves => L_Manifold_Valves,
        VO_Manifold_Pumps => L_Manifold_Pumps,
        VO_Zone_Valves => L_Zone_Valves,
        VO_Boiler_OT_Enable => L_Boiler_OT_Enable,
        VO_Boiler_OT_Setpoint => L_Boiler_OT_Setpoint,
        VO_Backup_Circulation_Pump => L_Backup_Circulation_Pump,
        VO_Electric_Heater_Enable => L_Electric_Heater_Enable,
        VO_Freeze_Risk_Status => L_Freeze_Risk_Status,
        VO_Status => L_Manifold_Status,
        VO_Boiler_Status => L_Boiler_Status
    );

    L_Runtime_Context.Heating_Executed := TRUE;

END_IF;

L_Runtime_Context.Current_Phase := E_Heating_Runtime_Phase.HRP_SERVICE_GATING;

fbServiceGatingPhase(
    VI_Enable := TRUE,
    VIO_Manifold_Pumps := L_Manifold_Pumps,
    VIO_Backup_Circulation_Pump := L_Backup_Circulation_Pump,
    VIO_Electric_Heater_Enable := L_Electric_Heater_Enable,
    VIO_DHW_Heating_Pump := L_DHW_Heating_Pump,
    VIO_DHW_Circ_Pump := L_DHW_Circ_Pump,
    VIO_DHW_Status := L_DHW_Status,
    VIO_Freeze_Risk_Status := L_Freeze_Risk_Status
);

L_Runtime_Context.Service_Gating_Executed := fbServiceGatingPhase.VO_Executed;
L_Runtime_Context.Safety_Isolation_Valid := fbServiceGatingPhase.VO_Valid;

L_Runtime_Context.Current_Phase := E_Heating_Runtime_Phase.HRP_STATE_PUBLICATION;

fbStatePublicationPhase(
    VI_Enable := TRUE,
    VI_Zone_Valves := L_Zone_Valves,
    VI_Manifold_Pumps := L_Manifold_Pumps,
    VI_Manifold_Valves := L_Manifold_Valves,
    VI_Boiler_OT_Enable := L_Boiler_OT_Enable,
    VI_Boiler_OT_Setpoint := L_Boiler_OT_Setpoint,
    VI_Backup_Circulation_Pump := L_Backup_Circulation_Pump,
    VI_Electric_Heater_Enable := L_Electric_Heater_Enable,
    VI_Freeze_Risk_Status := L_Freeze_Risk_Status,
    VI_Manifold_Status := L_Manifold_Status,
    VI_Boiler_Status := L_Boiler_Status,
    VI_DHW_Heating_Pump := L_DHW_Heating_Pump,
    VI_DHW_Circ_Pump := L_DHW_Circ_Pump,
    VI_DHW_Status := L_DHW_Status
);

L_Runtime_Context.State_Publication_Executed := fbStatePublicationPhase.VO_Executed;
L_Runtime_Context.State_Publication_Before_Diagnostics_Valid := fbStatePublicationPhase.VO_Valid;

L_Runtime_Context.Current_Phase := E_Heating_Runtime_Phase.HRP_DIAGNOSTICS;

fbDiagnosticsPhase(
    VI_Enable := TRUE,
    VI_System_Time_MS := GVL_STATUS.G_System_Time_MS
);

L_Runtime_Context.Diagnostics_Executed := fbDiagnosticsPhase.VO_Executed;
L_Runtime_Context.Diagnostics_Isolation_Valid := fbDiagnosticsPhase.VO_Valid;

fbObserverPhase(
    VI_Authorization_Stage := FALSE,
    VI_Finalization_Stage := TRUE,
    VI_Runtime_Context := L_Runtime_Context,
    VI_Diagnostics_Valid := L_Runtime_Context.Diagnostics_Isolation_Valid
);

fbMetaSupervisionPublisher(
    VI_Enable := TRUE,
    VI_Runtime_Observation_Valid := GVL_Heating_Runtime_Observation.G_Runtime_Observation_Valid,
    VI_Runtime_Observer_Ready := GVL_Heating_Runtime_Observation.G_Runtime_Observer_Ready,
    VI_Runtime_Observer_Fault := GVL_Heating_Runtime_Observation.G_Runtime_Observer_Fault,
    VI_Runtime_Status_Code := GVL_Heating_Runtime_Observation.G_Runtime_Observation_Status_Code,
    VI_Runtime_Status_Text := GVL_Heating_Runtime_Observation.G_Runtime_Observation_Status_Text
);

GVL_Heating_Runtime_Meta.G_Runtime_Meta_Supervision :=
    fbMetaSupervisionPublisher.VO_Meta;

GVL_Heating_Runtime_Meta.G_Runtime_Meta_Publication_Valid :=
    fbMetaSupervisionPublisher.VO_Publication_Valid;

GVL_Heating_Runtime_Meta.G_Runtime_Meta_Status_Code :=
    fbMetaSupervisionPublisher.VO_Meta.Status_Code;

GVL_Heating_Runtime_Meta.G_Runtime_Meta_Status_Text :=
    fbMetaSupervisionPublisher.VO_Meta.Status_Text;

fbExplainabilityPublisher(
    VI_Enable := TRUE,
    VI_System_Time_MS := GVL_STATUS.G_System_Time_MS,
    VI_Runtime_Context := L_Runtime_Context,
    VI_Runtime_Observation_Valid := GVL_Heating_Runtime_Observation.G_Runtime_Observation_Valid,
    VI_Runtime_Observer_Fault := GVL_Heating_Runtime_Observation.G_Runtime_Observer_Fault,
    VI_Runtime_Status_Code := GVL_Heating_Runtime_Observation.G_Runtime_Observation_Status_Code,
    VI_Runtime_Status_Text := GVL_Heating_Runtime_Observation.G_Runtime_Observation_Status_Text
);

GVL_Heating_Runtime_Explainability.G_Runtime_Phase_Event :=
    fbExplainabilityPublisher.VO_Phase_Event;

GVL_Heating_Runtime_Explainability.G_Runtime_Anomaly :=
    fbExplainabilityPublisher.VO_Anomaly;

GVL_Heating_Runtime_Explainability.G_Runtime_Blackbox_Event :=
    fbExplainabilityPublisher.VO_Blackbox_Event;

GVL_Heating_Runtime_Explainability.G_Runtime_Blackbox_Timeline :=
    fbExplainabilityPublisher.VO_Blackbox_Timeline;

GVL_Heating_Runtime_Explainability.G_Runtime_Event_Buffer :=
    fbExplainabilityPublisher.VO_Event_Buffer;

GVL_Heating_Runtime_Explainability.G_Runtime_Adaptive_Intelligence :=
    fbExplainabilityPublisher.VO_Adaptive_Intelligence;

GVL_Heating_Runtime_Explainability.G_Runtime_Causality_Graph :=
    fbExplainabilityPublisher.VO_Causality_Graph;

GVL_Heating_Runtime_Explainability.G_Runtime_Explainability_Publication_Valid :=
    fbExplainabilityPublisher.VO_Publication_Valid;

GVL_Heating_Runtime_Explainability.G_Runtime_Explainability_Status_Code :=
    fbExplainabilityPublisher.VO_Phase_Event.Status_Code;

GVL_Heating_Runtime_Explainability.G_Runtime_Explainability_Status_Text :=
    fbExplainabilityPublisher.VO_Phase_Event.Status_Text;

IF L_Distributed_Projection_Allowed THEN

    L_Runtime_Context.Current_Phase := E_Heating_Runtime_Phase.HRP_OUTPUT_PROJECTION;

    fbOutputProjectionPhase(
        VI_Enable := TRUE,
        VI_Zone_Valves := L_Zone_Valves,
        VI_Manifold_Pumps := L_Manifold_Pumps,
        VI_Manifold_Valves := L_Manifold_Valves,
        VI_DHW_Heating_Pump := L_DHW_Heating_Pump,
        VI_DHW_Circ_Pump := L_DHW_Circ_Pump,
        VI_Backup_Circulation_Pump := L_Backup_Circulation_Pump,
        VI_Electric_Heater_Enable := L_Electric_Heater_Enable
    );

    L_Runtime_Context.Output_Projection_Executed :=
        fbOutputProjectionPhase.VO_Executed;

    L_Runtime_Context.Output_Projection_Last_Valid :=
        fbOutputProjectionPhase.VO_Valid;

END_IF;

L_Runtime_Context.Current_Phase := E_Heating_Runtime_Phase.HRP_COMPLETE;

// >>> BULK_SYNC_ANCHOR: PRG_Heating <<<
END_PROGRAM

(* ---- PRG_Heating_Config_Defaults.st ---- *)
PROGRAM PRG_Heating_Config_Defaults
VAR
    L_i : INT;
    L_Manifold : BYTE;
END_VAR

// Default per-circuit comfort/economy profiles.
// This initializer only fills empty records and does not overwrite HMI-edited
// records after circuit_id has been assigned.
FOR L_i := 1 TO GVL_CONSTANTS.C_MAX_HEATING_CIRCUITS DO
    IF GVL_CONFIG.G_HMI_FloorHeating_Configs[L_i].circuit_id = 0 THEN
        CASE L_i OF
            1, 2, 3, 4:
                L_Manifold := 1;
            5, 6, 7, 8:
                L_Manifold := 2;
            9, 10, 11, 12:
                L_Manifold := 3;
            13, 14:
                L_Manifold := 4;
        ELSE
                L_Manifold := 5;
        END_CASE;

        GVL_CONFIG.G_HMI_FloorHeating_Configs[L_i].circuit_id := TO_BYTE(L_i);
        GVL_CONFIG.G_HMI_FloorHeating_Configs[L_i].zone := TO_BYTE(L_i);
        GVL_CONFIG.G_HMI_FloorHeating_Configs[L_i].manifold_id := L_Manifold;
        GVL_CONFIG.G_HMI_FloorHeating_Configs[L_i].sensor_id := TO_BYTE(L_i);
        GVL_CONFIG.G_HMI_FloorHeating_Configs[L_i].valve_id := TO_BYTE(L_i);
        GVL_CONFIG.G_HMI_FloorHeating_Configs[L_i].control_type := 1;

        // Historical design_temp is kept, but explicit comfort_temp is now the
        // room comfort setpoint used by FB_Heating_Circuit_Control.
        GVL_CONFIG.G_HMI_FloorHeating_Configs[L_i].design_temp := 22.0;
        GVL_CONFIG.G_HMI_FloorHeating_Configs[L_i].use_in_normal := TRUE;
        GVL_CONFIG.G_HMI_FloorHeating_Configs[L_i].use_in_away_preheat := TRUE;
        GVL_CONFIG.G_HMI_FloorHeating_Configs[L_i].comfort_temp := 22.0;
        GVL_CONFIG.G_HMI_FloorHeating_Configs[L_i].economy_temp := 17.0;
        GVL_CONFIG.G_HMI_FloorHeating_Configs[L_i].long_away_temp := 12.0;

        GVL_CONFIG.G_HMI_FloorHeating_Configs[L_i].min_temp := 5.0;
        GVL_CONFIG.G_HMI_FloorHeating_Configs[L_i].max_temp := 30.0;
        GVL_CONFIG.G_HMI_FloorHeating_Configs[L_i].pid_kp := 2.0;
        GVL_CONFIG.G_HMI_FloorHeating_Configs[L_i].pwm_period_s := 600;
    END_IF;
END_FOR;

END_PROGRAM

(* ---- PRG_Heating_Policy_Manager.st ---- *)
PROGRAM PRG_Heating_Policy_Manager

VAR
    fbPolicyManager : FB_Heating_Policy_Manager;
END_VAR

fbPolicyManager(
    VI_System_Mode := GVL_STATE.G_System_Mode,
    VI_RootCause := GVL_STATE.G_Heating_RootCause,
    VI_Emergency_Stop := GVL_STATE.G_Safety_Emergency_Stop,
    VI_Gas_Safety := GVL_STATE.G_Safety_Gas_Latched
);

GVL_HEATING_POLICY.G_Policy_Mode := fbPolicyManager.VO_Policy_Mode;
GVL_HEATING_POLICY.G_Policy_Block_Heating_Request := fbPolicyManager.VO_Block_Heating;

(* ---- PRG_Heating_Policy_Observer.st ---- *)
PROGRAM PRG_Heating_Policy_Observer
VAR
    fbPolicy : FB_Heating_Policy_Observer;
END_VAR

fbPolicy(
    VI_Zone_Occupied := GVL_PRESENCE.G_Zone_Occupied,
    VI_Zone_Last_Motion_TS := GVL_PRESENCE.G_Zone_Last_Motion_TS,
    VI_System_Time_MS := GVL_STATUS.G_System_Time_MS,
    VI_Zone_Permanent_Use := GVL_HEATING_POLICY.G_Zone_Permanent_Use,
    VI_Zone_Guest_Preheat := GVL_HEATING_POLICY.G_Zone_Guest_Preheat_Request,
    VI_Behavior_Mode := GVL_MODE.G_Current_Behavior_Mode
);

GVL_HEATING_POLICY.G_Zone_Empty_Duration_MS := fbPolicy.VO_Zone_Empty_Duration_MS;
GVL_HEATING_POLICY.G_Zone_Policy_Class := fbPolicy.VO_Zone_Policy_Class;
GVL_HEATING_POLICY.G_Zone_Target_Adjustment := fbPolicy.VO_Zone_Target_Adjustment;
GVL_HEATING_POLICY.G_Zone_Priority_Bias := fbPolicy.VO_Zone_Priority_Bias;
END_PROGRAM

(* ---- PRG_Heating_Supervisory_Publication.st ---- *)
PROGRAM PRG_Heating_Supervisory_Publication
VAR
    fbCircuitExplainabilityAdapter : FB_Heating_Circuit_Explainability_Adapter;
    fbSourceStabilityObserver : FB_Heating_Source_Stability_Observer;
    fbSupervisoryEnrichment : FB_Heating_Runtime_Supervisory_Enrichment;
    fbSupervisoryPublicationAdapter : FB_Heating_Runtime_Supervisory_Publication_Adapter;

    L_i : INT;
    L_Cascade_Boiler_Count : UINT;
    L_OT_Command_Valid : BOOL;
    L_Causality_Node : ST_Heating_Runtime_Causality_Node;
    L_Causality_Edge : ST_Heating_Runtime_Causality_Edge;
    L_Blackbox_Event : ST_Heating_Runtime_Blackbox_Event;
    L_Predictive_State : ST_Heating_Runtime_Predictive_State;
    L_Status_Code : UINT;
    L_Status_Text : STRING(128);
END_VAR

// ==============================================================================
// Heating supervisory publication orchestration
//
// Observation-only program.
// Runs after PRG_Heating has produced canonical runtime projection.
// Does not own runtime, outputs, commands or heating authority.
// ==============================================================================

// Compatibility publication from canonical runtime projection.
fbCircuitExplainabilityAdapter(
    VI_Enable := TRUE
);

// Per-circuit predictive source-stability observation from canonical projection.
fbSourceStabilityObserver(
    VI_Enable := TRUE,
    VI_System_Time_MS := GVL_STATUS.G_System_Time_MS
);

// Lightweight OT/cascade observation for supervisory enrichment context.
L_Cascade_Boiler_Count := 0;
L_OT_Command_Valid := TRUE;

FOR L_i := 1 TO GVL_CONSTANTS.C_MAX_BOILERS DO
    IF GVL_STATE.G_Boiler_OT_Online[L_i] THEN
        L_Cascade_Boiler_Count := L_Cascade_Boiler_Count + 1;
    END_IF;

    IF GVL_STATE.G_Boiler_OT_Enable[L_i] AND NOT GVL_STATE.G_Boiler_OT_Online[L_i] THEN
        L_OT_Command_Valid := FALSE;
    END_IF;
END_FOR;

// Supervisory enrichment owns timeline/event/reconstruction ingestion.
fbSupervisoryEnrichment(
    VI_Enable := TRUE,
    VI_System_Time_MS := GVL_STATUS.G_System_Time_MS,
    VI_Runtime_Context := GVL_Heating_Runtime_Observation.G_Runtime_Context,
    VI_Phase_Event := GVL_Heating_Runtime_Explainability.G_Runtime_Phase_Event,
    VI_Anomaly := GVL_Heating_Runtime_Explainability.G_Runtime_Anomaly,
    VI_Cascade_Boiler_Count := L_Cascade_Boiler_Count,
    VI_OT_Command_Valid := L_OT_Command_Valid,
    VIO_Event_Buffer := GVL_Heating_Runtime_Explainability.G_Runtime_Event_Buffer,
    VIO_Execution_Timeline := GVL_Heating_Runtime_Explainability.G_Runtime_Execution_Timeline,
    VO_Causality_Node => L_Causality_Node,
    VO_Causality_Edge => L_Causality_Edge,
    VO_Blackbox_Event => L_Blackbox_Event,
    VO_Predictive_State => L_Predictive_State,
    VO_Status_Code => L_Status_Code,
    VO_Status_Text => L_Status_Text
);

// Canonical supervisory publication surface.
fbSupervisoryPublicationAdapter(
    VI_Enable := TRUE,
    VI_Predictive_State := L_Predictive_State,
    VI_Causality_Node := L_Causality_Node,
    VI_Causality_Edge := L_Causality_Edge,
    VI_Blackbox_Event := L_Blackbox_Event,
    VI_Anomaly := GVL_Heating_Runtime_Explainability.G_Runtime_Anomaly
);

// Keep existing runtime explainability GVL as a compatibility publication surface.
GVL_Heating_Runtime_Explainability.G_Runtime_Blackbox_Event := L_Blackbox_Event;
GVL_Heating_Runtime_Explainability.G_Runtime_Predictive_State := L_Predictive_State;
GVL_Heating_Runtime_Explainability.G_Runtime_Explainability_Publication_Valid := TRUE;
GVL_Heating_Runtime_Explainability.G_Runtime_Explainability_Status_Code := L_Status_Code;
GVL_Heating_Runtime_Explainability.G_Runtime_Explainability_Status_Text := L_Status_Text;

// >>> BULK_SYNC_ANCHOR: PRG_Heating_Supervisory_Publication <<<
END_PROGRAM

(* ---- PRG_Historical_Truth_Governor.st ---- *)
PROGRAM PRG_Historical_Truth_Governor
VAR
    L_Now_MS : UDINT;
    L_History_Valid : BOOL := TRUE;
    L_Error_Code : UDINT := 0;
    L_Error_Text : STRING(160) := '';
END_VAR

L_Now_MS := GVL_STATUS.G_System_Time_MS;
L_History_Valid := TRUE;
L_Error_Code := 0;
L_Error_Text := '';

// Fail-safe defaults.
GVL_HISTORICAL_TRUTH.Historical_Truth_Valid := FALSE;
GVL_HISTORICAL_TRUTH.Historical_Truth_Granted := FALSE;
GVL_HISTORICAL_TRUTH.Historical_Truth_Quarantine_Active := TRUE;

GVL_HISTORICAL_TRUTH.Trend_History_Causally_Immutable := FALSE;
GVL_HISTORICAL_TRUTH.Alarm_Chronology_Immutable := FALSE;
GVL_HISTORICAL_TRUTH.Blackbox_Snapshot_Immutable := FALSE;
GVL_HISTORICAL_TRUTH.Diagnostics_History_Coherent := FALSE;
GVL_HISTORICAL_TRUTH.Failover_Chronology_Coherent := FALSE;

// Observability truth authority required.
IF NOT GVL_OBSERVABILITY_TRUTH.Observability_Truth_Granted THEN
    L_History_Valid := FALSE;
    L_Error_Code := 33000;
    L_Error_Text := 'Observability truth authority not granted';
END_IF;

// Historical corruption detectors.
IF GVL_HISTORICAL_TRUTH.History_Epoch_Skew_Detected THEN
    L_History_Valid := FALSE;
    L_Error_Code := 33001;
    L_Error_Text := 'Historical epoch skew detected';
END_IF;

IF GVL_HISTORICAL_TRUTH.Failover_Chronology_Corruption_Detected THEN
    L_History_Valid := FALSE;
    L_Error_Code := 33002;
    L_Error_Text := 'Failover chronology corruption detected';
END_IF;

IF GVL_HISTORICAL_TRUTH.Trend_Replay_Race_Detected THEN
    L_History_Valid := FALSE;
    L_Error_Code := 33003;
    L_Error_Text := 'Trend replay race detected';
END_IF;

IF GVL_HISTORICAL_TRUTH.Blackbox_Causality_Drift_Detected THEN
    L_History_Valid := FALSE;
    L_Error_Code := 33004;
    L_Error_Text := 'Blackbox causality drift detected';
END_IF;

IF GVL_HISTORICAL_TRUTH.Alarm_Order_Reconstruction_Error THEN
    L_History_Valid := FALSE;
    L_Error_Code := 33005;
    L_Error_Text := 'Alarm order reconstruction error detected';
END_IF;

IF GVL_HISTORICAL_TRUTH.Mixed_Authority_Persistence_Detected THEN
    L_History_Valid := FALSE;
    L_Error_Code := 33006;
    L_Error_Text := 'Mixed-authority persistence detected';
END_IF;

// Historical persistence integrity validation.
IF L_History_Valid
AND NOT GVL_HISTORICAL_TRUTH.Persisted_Epochs_Coherent THEN
    L_History_Valid := FALSE;
    L_Error_Code := 33010;
    L_Error_Text := 'Persisted epoch coherence invalid';
END_IF;

IF L_History_Valid
AND NOT GVL_HISTORICAL_TRUTH.Recovery_Replay_Coherent THEN
    L_History_Valid := FALSE;
    L_Error_Code := 33011;
    L_Error_Text := 'Recovery replay coherence invalid';
END_IF;

IF L_History_Valid
AND NOT GVL_HISTORICAL_TRUTH.Historical_Snapshot_Coherent THEN
    L_History_Valid := FALSE;
    L_Error_Code := 33012;
    L_Error_Text := 'Historical snapshot coherence invalid';
END_IF;

IF L_History_Valid
AND NOT GVL_HISTORICAL_TRUTH.Mixed_Authority_Persistence_Absent THEN
    L_History_Valid := FALSE;
    L_Error_Code := 33013;
    L_Error_Text := 'Mixed-authority persistence absence invalid';
END_IF;

IF L_History_Valid THEN
    GVL_HISTORICAL_TRUTH.Historical_Truth_Valid := TRUE;
    GVL_HISTORICAL_TRUTH.Historical_Truth_Granted := TRUE;
    GVL_HISTORICAL_TRUTH.Historical_Truth_Quarantine_Active := FALSE;

    GVL_HISTORICAL_TRUTH.Trend_History_Causally_Immutable := TRUE;
    GVL_HISTORICAL_TRUTH.Alarm_Chronology_Immutable := TRUE;
    GVL_HISTORICAL_TRUTH.Blackbox_Snapshot_Immutable := TRUE;
    GVL_HISTORICAL_TRUTH.Diagnostics_History_Coherent := TRUE;
    GVL_HISTORICAL_TRUTH.Failover_Chronology_Coherent := TRUE;

    GVL_HISTORICAL_TRUTH.Historical_Truth_Epoch :=
        GVL_OBSERVABILITY_TRUTH.Observability_Truth_Epoch;

    GVL_HISTORICAL_TRUTH.Historical_Truth_Epoch_Coherent := TRUE;

    GVL_HISTORICAL_TRUTH.Historical_Last_Update_MS := L_Now_MS;
    GVL_HISTORICAL_TRUTH.Historical_Lease_Expired := FALSE;

    GVL_HISTORICAL_TRUTH.Historical_Last_Error_Code := 0;
    GVL_HISTORICAL_TRUTH.Historical_Last_Error_Text := '';
ELSE
    GVL_HISTORICAL_TRUTH.Historical_Truth_Valid := FALSE;
    GVL_HISTORICAL_TRUTH.Historical_Truth_Granted := FALSE;
    GVL_HISTORICAL_TRUTH.Historical_Truth_Quarantine_Active := TRUE;

    GVL_HISTORICAL_TRUTH.Historical_Lease_Expired := TRUE;

    GVL_HISTORICAL_TRUTH.Historical_Last_Error_Code :=
        L_Error_Code;

    GVL_HISTORICAL_TRUTH.Historical_Last_Error_Text :=
        L_Error_Text;

    GVL_HISTORICAL_TRUTH.Historical_Invalidation_Count :=
        GVL_HISTORICAL_TRUTH.Historical_Invalidation_Count + 1;
END_IF;

END_PROGRAM

(* ---- PRG_HMI_Access_Dashboard.st ---- *)
PROGRAM PRG_HMI_Access_Dashboard

GVL_HMI_ACCESS.G_Safety_Mode := GVL_SAFETY_SHUTDOWN.G_Safety_Mode;
GVL_HMI_ACCESS.G_User_Access_Level := GVL_INTENT_USER.I_User_Access_Level;
GVL_HMI_ACCESS.G_Manual_Access_OK :=
    GVL_INTENT_USER.I_Source_Valid AND (GVL_INTENT_USER.I_User_Access_Level >= 2);

GVL_HMI_ACCESS.G_Runtime_Required := GVL_ACCESS_RUNTIME.G_Runtime_Required;
GVL_HMI_ACCESS.G_Runtime_Executed := GVL_ACCESS_RUNTIME.G_Runtime_Executed;
GVL_HMI_ACCESS.G_Runtime_Idle_By_Design := GVL_ACCESS_RUNTIME.G_Runtime_Idle_By_Design;
GVL_HMI_ACCESS.G_Runtime_Blocked_By_Distributed_Gates := GVL_ACCESS_RUNTIME.G_Runtime_Blocked_By_Distributed_Gates;
GVL_HMI_ACCESS.G_Any_Pulse_Active := GVL_ACCESS_RUNTIME.G_Any_Pulse_Active;
GVL_HMI_ACCESS.G_Last_Update_MS := GVL_ACCESS_RUNTIME.G_Last_Update_MS;
GVL_HMI_ACCESS.G_Status_Code := GVL_ACCESS_RUNTIME.G_Status_Code;
GVL_HMI_ACCESS.G_Status_Text := GVL_ACCESS_RUNTIME.G_Status_Text;

GVL_HMI_ACCESS.G_Command_Lock_1_Open := GVL_COMMAND_SHADOW.G_Lock_1_Open;
GVL_HMI_ACCESS.G_Command_Lock_1_Close := GVL_COMMAND_SHADOW.G_Lock_1_Close;
GVL_HMI_ACCESS.G_Command_Lock_2_Open := GVL_COMMAND_SHADOW.G_Lock_2_Open;
GVL_HMI_ACCESS.G_Command_Lock_2_Close := GVL_COMMAND_SHADOW.G_Lock_2_Close;
GVL_HMI_ACCESS.G_Command_Gate_Open := GVL_COMMAND_SHADOW.G_Gate_Open;
GVL_HMI_ACCESS.G_Command_Wicket_Open := GVL_COMMAND_SHADOW.G_Wicket_Open;

GVL_HMI_ACCESS.G_Output_Lock_1_Open := GVL_ACCESS_OUTPUT.DO_Lock_1_Open;
GVL_HMI_ACCESS.G_Output_Lock_1_Close := GVL_ACCESS_OUTPUT.DO_Lock_1_Close;
GVL_HMI_ACCESS.G_Output_Lock_2_Open := GVL_ACCESS_OUTPUT.DO_Lock_2_Open;
GVL_HMI_ACCESS.G_Output_Lock_2_Close := GVL_ACCESS_OUTPUT.DO_Lock_2_Close;
GVL_HMI_ACCESS.G_Output_Gate_Open := GVL_ACCESS_OUTPUT.DO_Gate_Open;
GVL_HMI_ACCESS.G_Output_Wicket_Open := GVL_ACCESS_OUTPUT.DO_Wicket_Open;

GVL_HMI_ACCESS.G_Physical_Lock_1_Open := GVL_IO.DO_Lock_1_Open;
GVL_HMI_ACCESS.G_Physical_Lock_1_Close := GVL_IO.DO_Lock_1_Close;
GVL_HMI_ACCESS.G_Physical_Lock_2_Open := GVL_IO.DO_Lock_2_Open;
GVL_HMI_ACCESS.G_Physical_Lock_2_Close := GVL_IO.DO_Lock_2_Close;
GVL_HMI_ACCESS.G_Physical_Gate_Open := GVL_IO.DO_Gate_Open;
GVL_HMI_ACCESS.G_Physical_Wicket_Open := GVL_IO.DO_Wicket_Open;

GVL_HMI_ACCESS.G_Fire_Evacuation_Access_Active := GVL_SAFETY_SHUTDOWN.G_Safety_Mode = FIRE;
GVL_HMI_ACCESS.G_Gas_Access_Release_Active := GVL_SAFETY_SHUTDOWN.G_Safety_Mode = GAS;
GVL_HMI_ACCESS.G_Safety_Cleared_Active :=
    (GVL_SAFETY_SHUTDOWN.G_Safety_Mode = WATER_LEAK)
    OR (GVL_SAFETY_SHUTDOWN.G_Safety_Mode = GLOBAL_STOP);
GVL_HMI_ACCESS.G_Distributed_Block_Active := GVL_ACCESS_RUNTIME.G_Runtime_Blocked_By_Distributed_Gates;

IF GVL_HMI_ACCESS.G_Fire_Evacuation_Access_Active THEN
    GVL_HMI_ACCESS.G_Reason_Text := 'Fire evacuation access active';
ELSIF GVL_HMI_ACCESS.G_Gas_Access_Release_Active THEN
    GVL_HMI_ACCESS.G_Reason_Text := 'Gas access release active';
ELSIF GVL_HMI_ACCESS.G_Safety_Cleared_Active THEN
    GVL_HMI_ACCESS.G_Reason_Text := 'Access outputs cleared by safety mode';
ELSIF GVL_HMI_ACCESS.G_Distributed_Block_Active THEN
    GVL_HMI_ACCESS.G_Reason_Text := 'Access blocked by distributed gates';
ELSIF GVL_HMI_ACCESS.G_Any_Pulse_Active THEN
    GVL_HMI_ACCESS.G_Reason_Text := 'Access pulse active';
ELSIF GVL_HMI_ACCESS.G_Manual_Access_OK THEN
    GVL_HMI_ACCESS.G_Reason_Text := 'Manual access allowed';
ELSE
    GVL_HMI_ACCESS.G_Reason_Text := 'Access idle or manual access denied';
END_IF;

// >>> BULK_SYNC_ANCHOR: PRG_HMI_Access_Dashboard <<<
END_PROGRAM

(* ---- PRG_HMI_Alarm_Audible_Ack_Dashboard.st ---- *)
PROGRAM PRG_HMI_Alarm_Audible_Ack_Dashboard

GVL_HMI_ALARM_AUDIBLE_ACK.G_Ack_Active := GVL_ALARM_AUDIBLE_ACK.G_Ack_Active;
GVL_HMI_ALARM_AUDIBLE_ACK.G_Ack_Remaining_MS := GVL_ALARM_AUDIBLE_ACK.G_Ack_Remaining_MS;
GVL_HMI_ALARM_AUDIBLE_ACK.G_Ack_Count_Current_Alarm := GVL_ALARM_AUDIBLE_ACK.G_Ack_Count_Current_Alarm;
GVL_HMI_ALARM_AUDIBLE_ACK.G_Ack_Limit_Reached := GVL_ALARM_AUDIBLE_ACK.G_Ack_Limit_Reached;
GVL_HMI_ALARM_AUDIBLE_ACK.G_Last_Ack_Accepted := GVL_ALARM_AUDIBLE_ACK.G_Last_Ack_Accepted;
GVL_HMI_ALARM_AUDIBLE_ACK.G_Last_Ack_Denied := GVL_ALARM_AUDIBLE_ACK.G_Last_Ack_Denied;
GVL_HMI_ALARM_AUDIBLE_ACK.G_Last_Denial_Code := GVL_ALARM_AUDIBLE_ACK.G_Last_Denial_Code;
GVL_HMI_ALARM_AUDIBLE_ACK.G_Last_Event_MS := GVL_ALARM_AUDIBLE_ACK.G_Last_Event_MS;
GVL_HMI_ALARM_AUDIBLE_ACK.G_Status_Text := GVL_ALARM_AUDIBLE_ACK.G_Status_Text;
GVL_HMI_ALARM_AUDIBLE_ACK.G_Effective_Siren_Muted := GVL_ALARM_AUDIBLE_ACK.G_Ack_Active;

// >>> BULK_SYNC_ANCHOR: PRG_HMI_Alarm_Audible_Ack_Dashboard <<<
END_PROGRAM

(* ---- PRG_HMI_Config_Workflow_Manager.st ---- *)
PROGRAM PRG_HMI_Config_Workflow_Manager
// ==============================================================================
// HMI CONFIG WORKFLOW MANAGER — runtime bridge for operator config workflow.
// ==============================================================================
// Runs config activation, HMI workflow and staged-config simulation. The activation
// FB refreshes staged topology state first; the workflow FB publishes simulation
// and config-control requests; simulation then consumes validation requests.
// ==============================================================================
VAR
    fbHMIConfigWorkflow : FB_HMI_Config_Workflow_Runtime;
    fbConfigActivation : FB_Config_Activation_Runtime;
    fbConfigSimulation : FB_Config_Simulation;
END_VAR

fbConfigActivation(
    VI_Enable := TRUE,
    VI_System_Time_MS := GVL_TIME_SERVICE.G_Now_MS
);

fbHMIConfigWorkflow(
    VI_Enable := TRUE,
    VI_System_Time_MS := GVL_TIME_SERVICE.G_Now_MS
);

fbConfigSimulation(
    VI_Enable := TRUE,
    VI_Request := GVL_CONFIG_SIMULATION.G_Simulation_Request,
    VI_Confirm := GVL_CONFIG_SIMULATION.G_Simulation_Confirm
);

// >>> BULK_SYNC_ANCHOR: PRG_HMI_Config_Workflow_Manager <<<
END_PROGRAM

(* ---- PRG_HMI_Dashboard.st ---- *)
PROGRAM PRG_HMI_Dashboard
VAR
    L_i : INT;
    L_Archive_Target_Available : BOOL;
END_VAR

// ======================================================
// HEATING CONFIDENCE
// ======================================================
GVL_HMI.G_HMI_Heating_Confidence := GVL_STATE.G_Heating_Confidence;
GVL_HMI.G_HMI_Heating_Confidence_Percent := REAL_TO_INT(GVL_STATE.G_Heating_Confidence * 100.0);

// ======================================================
// HEATING ROOT CAUSE
// ======================================================
GVL_HMI.G_HMI_Heating_Reason_Code := GVL_STATE.G_Heating_Confidence_Reason_Code;
GVL_HMI.G_HMI_Heating_Status_Text := GVL_STATE.G_Heating_Confidence_Reason_Text;

// ======================================================
// HEATING STATUS LEVEL
// ======================================================
IF GVL_STATE.G_Heating_Confidence > 0.8 THEN
    GVL_HMI.G_HMI_Heating_Status_Level := 0;
ELSIF GVL_STATE.G_Heating_Confidence > 0.5 THEN
    GVL_HMI.G_HMI_Heating_Status_Level := 1;
ELSE
    GVL_HMI.G_HMI_Heating_Status_Level := 2;
END_IF;

// ======================================================
// CASCADE SEMANTIC STATE
// ======================================================
GVL_HMI.G_HMI_Heating_Cascade_Available :=
    GVL_STATE.G_Heating_Cascade_Available;

GVL_HMI.G_HMI_Heating_Cascade_Degraded :=
    GVL_STATE.G_Heating_Cascade_Degraded;

GVL_HMI.G_HMI_Heating_Cascade_Partial_Capacity :=
    GVL_STATE.G_Heating_Cascade_Partial_Capacity;

GVL_HMI.G_HMI_Heating_Cascade_No_Flame :=
    GVL_STATE.G_Heating_Cascade_No_Flame;

GVL_HMI.G_HMI_Heating_Cascade_Transport_Degraded :=
    GVL_STATE.G_Heating_Cascade_Transport_Degraded;

GVL_HMI.G_HMI_Heating_Cascade_Ignition_Timeout :=
    GVL_STATE.G_Heating_Cascade_Ignition_Timeout;

GVL_HMI.G_HMI_Heating_Cascade_Active_Boilers :=
    GVL_STATE.G_Heating_Cascade_Active_Boilers;

GVL_HMI.G_HMI_Heating_Cascade_Available_Boilers :=
    GVL_STATE.G_Heating_Cascade_Available_Boilers;

// ======================================================
// OPENTHERM SEMANTIC STATE
// ======================================================
FOR L_i := 1 TO GVL_CONSTANTS.C_MAX_BOILERS DO

    GVL_HMI.G_HMI_Boiler_OT_Online[L_i] :=
        GVL_STATE.G_Boiler_OT_Online[L_i];

    GVL_HMI.G_HMI_Boiler_OT_Command_Ack[L_i] :=
        GVL_STATE.G_Boiler_OT_Command_Ack[L_i];

    GVL_HMI.G_HMI_Boiler_OT_Command_Timeout[L_i] :=
        GVL_STATE.G_Boiler_OT_Command_Timeout[L_i];

    GVL_HMI.G_HMI_Boiler_OT_Heartbeat_Timeout[L_i] :=
        GVL_STATE.G_Boiler_OT_Heartbeat_Timeout[L_i];

    GVL_HMI.G_HMI_Boiler_OT_Adapter_Error[L_i] :=
        GVL_STATE.G_Boiler_OT_Adapter_Error[L_i];

    GVL_HMI.G_HMI_Boiler_OT_Heartbeat_Age_MS[L_i] :=
        GVL_STATE.G_Boiler_OT_Heartbeat_Age_MS[L_i];

    GVL_HMI.G_HMI_Boiler_OT_Command_Age_MS[L_i] :=
        GVL_STATE.G_Boiler_OT_Command_Age_MS[L_i];

    GVL_HMI.G_HMI_Boiler_OT_Adapter_State[L_i] :=
        GVL_STATE.G_Boiler_OT_Adapter_State[L_i];

    GVL_HMI.G_HMI_Boiler_OT_Error_State[L_i] :=
        GVL_STATE.G_Boiler_OT_Error_State[L_i];

END_FOR;

// ======================================================
// PREDICTIVE FLAGS
// ======================================================
FOR L_i := 1 TO GVL_CONSTANTS.C_MAX_MANIFOLDS DO
    GVL_HMI.G_HMI_Heating_Predictive_Pressure_Drop[L_i] :=
        GVL_STATE.G_Predictive_Pump_Pressure_Drop[L_i];

    GVL_HMI.G_HMI_Heating_Predictive_Current_Rise[L_i] :=
        GVL_STATE.G_Predictive_Pump_Current_Rise[L_i];
END_FOR;

// ======================================================
// FILE / ARCHIVE STATUS (READ-ONLY DASHBOARD)
// ======================================================
L_Archive_Target_Available := FALSE;
CASE GVL_FILE_ARCHIVE.G_File_Archive_Target_Code OF
    1:
        L_Archive_Target_Available := GVL_FILE_ARCHIVE.G_PLC_File_Target_Available;
    2:
        L_Archive_Target_Available := GVL_FILE_ARCHIVE.G_USB_Target_Available;
    3:
        L_Archive_Target_Available := GVL_FILE_ARCHIVE.G_Gateway_Target_Available;
ELSE
    L_Archive_Target_Available := FALSE;
END_CASE;

GVL_HMI.G_HMI_File_Archive_Interface_Enabled := GVL_FILE_ARCHIVE.G_Archive_Interface_Enabled;
GVL_HMI.G_HMI_File_Archive_CSV_Enabled := GVL_FILE_ARCHIVE.G_CSV_Write_Enabled;
GVL_HMI.G_HMI_File_Archive_Target_Code := GVL_FILE_ARCHIVE.G_File_Archive_Target_Code;
GVL_HMI.G_HMI_File_Archive_Target_Available := L_Archive_Target_Available;
GVL_HMI.G_HMI_File_Archive_Write_Busy := GVL_FILE_ARCHIVE.G_Write_Busy;
GVL_HMI.G_HMI_File_Archive_Write_Done := GVL_FILE_ARCHIVE.G_Write_Done;
GVL_HMI.G_HMI_File_Archive_Write_Error := GVL_FILE_ARCHIVE.G_Write_Error;
GVL_HMI.G_HMI_File_Archive_Last_Error_Code := GVL_FILE_ARCHIVE.G_Last_Error_Code;
GVL_HMI.G_HMI_File_Archive_Last_Status_Text := GVL_FILE_ARCHIVE.G_Last_Status_Text;
GVL_HMI.G_HMI_File_Archive_Last_Write_MS := GVL_FILE_ARCHIVE.G_Last_Write_MS;

GVL_HMI.G_HMI_File_Archive_Auto_Backup_Enabled := GVL_FILE_ARCHIVE.G_Auto_Config_Backup_Enabled;
GVL_HMI.G_HMI_File_Archive_Auto_Backup_Time_Of_Day_MS := GVL_FILE_ARCHIVE.G_Auto_Config_Backup_Time_Of_Day_MS;
GVL_HMI.G_HMI_File_Archive_Auto_Backup_Last_Day_Of_Week := GVL_FILE_ARCHIVE.G_Auto_Config_Backup_Last_Day_Of_Week;
GVL_HMI.G_HMI_File_Archive_Auto_Backup_Last_Request_MS := GVL_FILE_ARCHIVE.G_Auto_Config_Backup_Last_Request_MS;
GVL_HMI.G_HMI_File_Archive_Auto_Backup_Last_Status_Text := GVL_FILE_ARCHIVE.G_Auto_Config_Backup_Last_Status_Text;

IF GVL_FILE_ARCHIVE.G_Write_Error THEN
    GVL_HMI.G_HMI_File_Archive_Status_Level := 2;
ELSIF GVL_FILE_ARCHIVE.G_Write_Busy THEN
    GVL_HMI.G_HMI_File_Archive_Status_Level := 1;
ELSIF GVL_FILE_ARCHIVE.G_Archive_Interface_Enabled AND GVL_FILE_ARCHIVE.G_CSV_Write_Enabled AND L_Archive_Target_Available THEN
    GVL_HMI.G_HMI_File_Archive_Status_Level := 0;
ELSE
    GVL_HMI.G_HMI_File_Archive_Status_Level := 1;
END_IF;

END_PROGRAM

(* ---- PRG_HMI_Gas_Smoke_CO_Dashboard.st ---- *)
PROGRAM PRG_HMI_Gas_Smoke_CO_Dashboard
VAR
    L_i : INT;
    L_Methane_Max : REAL;
    L_CO_Max : REAL;
    L_Smoke_Count : UINT;
END_VAR

L_Methane_Max := 0.0;
FOR L_i := 1 TO GVL_CONSTANTS.C_MAX_METHANE_SENSORS DO
    GVL_HMI_GAS_SMOKE_CO.G_Methane_Effective[L_i] := GVL_Safety_Selector.G_Methane_Effective_Array[L_i];
    IF GVL_Safety_Selector.G_Methane_Effective_Array[L_i] > L_Methane_Max THEN
        L_Methane_Max := GVL_Safety_Selector.G_Methane_Effective_Array[L_i];
    END_IF;
END_FOR;
GVL_HMI_GAS_SMOKE_CO.G_Methane_Max_LEL := L_Methane_Max;

L_CO_Max := 0.0;
FOR L_i := 1 TO GVL_CONSTANTS.C_MAX_CO_SENSORS DO
    GVL_HMI_GAS_SMOKE_CO.G_CO_Effective[L_i] := GVL_Safety_Selector.G_CO_Effective_Array[L_i];
    IF GVL_Safety_Selector.G_CO_Effective_Array[L_i] > L_CO_Max THEN
        L_CO_Max := GVL_Safety_Selector.G_CO_Effective_Array[L_i];
    END_IF;
END_FOR;
GVL_HMI_GAS_SMOKE_CO.G_CO_Max_PPM := L_CO_Max;

L_Smoke_Count := 0;
FOR L_i := 1 TO GVL_CONSTANTS.C_MAX_SMOKE_SENSORS DO
    GVL_HMI_GAS_SMOKE_CO.G_Smoke_Effective[L_i] := GVL_Safety_Selector.G_Smoke_Effective_Array[L_i];
    IF GVL_Safety_Selector.G_Smoke_Effective_Array[L_i] THEN
        L_Smoke_Count := L_Smoke_Count + 1;
    END_IF;
END_FOR;
GVL_HMI_GAS_SMOKE_CO.G_Smoke_Active_Count := L_Smoke_Count;

GVL_HMI_GAS_SMOKE_CO.G_Methane_Warning_Level := GVL_HEALTH_BRIDGE.G_Methane_Warning_Level;
GVL_HMI_GAS_SMOKE_CO.G_Methane_Alarm_Level := GVL_HEALTH_BRIDGE.G_Methane_Alarm_Level;
GVL_HMI_GAS_SMOKE_CO.G_Methane_Critical_Level := GVL_HEALTH_BRIDGE.G_Methane_Critical_Level;
GVL_HMI_GAS_SMOKE_CO.G_CO_Warning_Level := GVL_HEALTH_BRIDGE.G_CO_Warning_Level;
GVL_HMI_GAS_SMOKE_CO.G_CO_Alarm_Level := GVL_HEALTH_BRIDGE.G_CO_Alarm_Level;
GVL_HMI_GAS_SMOKE_CO.G_Smoke_Detected := GVL_HEALTH_BRIDGE.G_Smoke_Detected;
GVL_HMI_GAS_SMOKE_CO.G_Gas_Detected := GVL_HEALTH_BRIDGE.G_Gas_Detected;
GVL_HMI_GAS_SMOKE_CO.G_Status_Text := GVL_STATUS.G_Gas_Status_Msg;

GVL_HMI_GAS_SMOKE_CO.G_Safety_Fire_Alarm_Active := GVL_INTENT_SAFETY.I_Fire_Alarm_Active;
GVL_HMI_GAS_SMOKE_CO.G_Safety_Gas_Alarm_Active := GVL_INTENT_SAFETY.I_Gas_Alarm_Active;
GVL_HMI_GAS_SMOKE_CO.G_Safety_CO_Warning_Active := GVL_INTENT_SAFETY.I_CO_Warning_Active;
GVL_HMI_GAS_SMOKE_CO.G_Gas_Close_Required := GVL_INTENT_SAFETY.I_Gas_Close_Required;
GVL_HMI_GAS_SMOKE_CO.G_Boiler_Stop_Required := GVL_INTENT_SAFETY.I_Boiler_Stop_Required;
GVL_HMI_GAS_SMOKE_CO.G_System_Safe_Stop_Required := GVL_INTENT_SAFETY.I_System_Safe_Stop_Required;
GVL_HMI_GAS_SMOKE_CO.G_Evacuation_Mode_Active := GVL_INTENT_SAFETY.I_Evacuation_Mode_Active;
GVL_HMI_GAS_SMOKE_CO.G_Vent_Stop_Required := GVL_INTENT_SAFETY.I_Vent_Stop_Required;
GVL_HMI_GAS_SMOKE_CO.G_Vent_Force_PV3_Boost := GVL_INTENT_SAFETY.I_Vent_Force_PV3_Boost;
GVL_HMI_GAS_SMOKE_CO.G_Vent_Force_Supply_100 := GVL_INTENT_SAFETY.I_Vent_Force_Supply_100;
GVL_HMI_GAS_SMOKE_CO.G_Vent_Force_Supply_80 := GVL_INTENT_SAFETY.I_Vent_Force_Supply_80;
GVL_HMI_GAS_SMOKE_CO.G_Vent_Force_Exhaust_100 := GVL_INTENT_SAFETY.I_Vent_Force_Exhaust_100;

GVL_HMI_GAS_SMOKE_CO.G_Vent_Output_Enable := GVL_VENT_OUTPUT.DO_Vent_Enable;
FOR L_i := 1 TO GVL_CONSTANTS.C_MAX_SUPPLY_FANS DO
    GVL_HMI_GAS_SMOKE_CO.G_Vent_Output_Supply_Fans[L_i] := GVL_VENT_OUTPUT.AO_Supply_Fans[L_i];
END_FOR;
FOR L_i := 1 TO GVL_CONSTANTS.C_MAX_EXHAUST_FANS DO
    GVL_HMI_GAS_SMOKE_CO.G_Vent_Output_Exhaust_Fans[L_i] := GVL_VENT_OUTPUT.AO_Exhaust_Fans[L_i];
END_FOR;

IF GVL_HEALTH_BRIDGE.G_Methane_Critical_Level OR GVL_INTENT_SAFETY.I_System_Safe_Stop_Required THEN
    GVL_HMI_GAS_SMOKE_CO.G_Status_Level := 3;
ELSIF GVL_HEALTH_BRIDGE.G_Methane_Alarm_Level OR GVL_HEALTH_BRIDGE.G_CO_Alarm_Level OR GVL_HEALTH_BRIDGE.G_Smoke_Detected THEN
    GVL_HMI_GAS_SMOKE_CO.G_Status_Level := 2;
ELSIF GVL_HEALTH_BRIDGE.G_Methane_Warning_Level OR GVL_HEALTH_BRIDGE.G_CO_Warning_Level THEN
    GVL_HMI_GAS_SMOKE_CO.G_Status_Level := 1;
ELSE
    GVL_HMI_GAS_SMOKE_CO.G_Status_Level := 0;
END_IF;

// >>> BULK_SYNC_ANCHOR: PRG_HMI_Gas_Smoke_CO_Dashboard <<<
END_PROGRAM

(* ---- PRG_HMI_Security_Access_Intent_Dashboard.st ---- *)
PROGRAM PRG_HMI_Security_Access_Intent_Dashboard

GVL_HMI_SECURITY_ACCESS_INTENT.G_Close_Request := GVL_SECURITY_ACCESS_INTENT.G_Auto_Lock_Close_Request;
GVL_HMI_SECURITY_ACCESS_INTENT.G_Close_Accepted := GVL_SECURITY_ACCESS_INTENT.G_Auto_Lock_Close_Accepted_By_Arbitration;
GVL_HMI_SECURITY_ACCESS_INTENT.G_Last_Request_MS := GVL_SECURITY_ACCESS_INTENT.G_Last_Auto_Lock_Request_MS;
GVL_HMI_SECURITY_ACCESS_INTENT.G_Status_Text := GVL_SECURITY_ACCESS_INTENT.G_Status_Text;

// >>> BULK_SYNC_ANCHOR: PRG_HMI_Security_Access_Intent_Dashboard <<<
END_PROGRAM

(* ---- PRG_HMI_Security_Dashboard.st ---- *)
PROGRAM PRG_HMI_Security_Dashboard
VAR
    L_i : INT;
    L_Motion_Count : INT;
    L_Door_Count : INT;
    L_Window_Count : INT;
END_VAR

L_Motion_Count := 0;
L_Door_Count := 0;
L_Window_Count := 0;

GVL_HMI_SECURITY.G_Armed := GVL_ALARM.G_Security_Armed;
GVL_HMI_SECURITY.G_Alarm_Active := GVL_ALARM.G_Security_Alarm;
GVL_HMI_SECURITY.G_Siren_Request := GVL_ALARM.G_Security_Siren;
GVL_HMI_SECURITY.G_Security_Alarm := GVL_ALARM.G_Security_Alarm;
GVL_HMI_SECURITY.G_Security_Siren := GVL_ALARM.G_Security_Siren;
GVL_HMI_SECURITY.G_Global_Siren := GVL_ALARM.G_Global_Siren;
GVL_HMI_SECURITY.G_Status_Text := GVL_STATUS.G_Security_Status_Msg;
GVL_HMI_SECURITY.G_Arm_Request := GVL_INTENT_USER.I_Arm_Request;
GVL_HMI_SECURITY.G_Disarm_Request := GVL_INTENT_USER.I_Disarm_Request;
GVL_HMI_SECURITY.G_Send_2FA_Req := GVL_COMMAND.G_Send_2FA_Req;
GVL_HMI_SECURITY.G_Last_Update_MS := GVL_TIME_SERVICE.G_Now_MS;

GVL_HMI_SECURITY.G_Safety_Access_Active :=
    (GVL_SAFETY_SHUTDOWN.G_Safety_Mode = FIRE)
    OR (GVL_SAFETY_SHUTDOWN.G_Safety_Mode = GAS);
GVL_HMI_SECURITY.G_Sensor_Path_Suppressed_By_Safety := GVL_HMI_SECURITY.G_Safety_Access_Active;

IF GVL_HMI_SECURITY.G_Sensor_Path_Suppressed_By_Safety THEN
    GVL_HMI_SECURITY.G_Sensor_Path_Status_Text := 'Security sensors suppressed by safety access mode';
ELSE
    GVL_HMI_SECURITY.G_Sensor_Path_Status_Text := 'Security sensors active';
END_IF;

FOR L_i := 1 TO 16 DO
    GVL_HMI_SECURITY.G_Motion_Active[L_i] := GVL_STATE.G_Motion_Sensors[L_i];
    GVL_HMI_SECURITY.G_Motion_Bypass[L_i] := GVL_CONFIG.G_Security_Config.bypass_motion[L_i];

    IF GVL_STATE.G_Motion_Sensors[L_i] AND NOT GVL_CONFIG.G_Security_Config.bypass_motion[L_i] THEN
        L_Motion_Count := L_Motion_Count + 1;
    END_IF;
END_FOR;

FOR L_i := 1 TO GVL_CONSTANTS.C_MAX_DOOR_SENSORS DO
    GVL_HMI_SECURITY.G_Door_Active[L_i] := GVL_STATE.G_Door_Sensors[L_i];
    GVL_HMI_SECURITY.G_Door_Bypass[L_i] := GVL_CONFIG.G_Security_Config.bypass_doors[L_i];

    IF GVL_STATE.G_Door_Sensors[L_i] AND NOT GVL_CONFIG.G_Security_Config.bypass_doors[L_i] THEN
        L_Door_Count := L_Door_Count + 1;
    END_IF;
END_FOR;

FOR L_i := 1 TO 16 DO
    GVL_HMI_SECURITY.G_Window_Active[L_i] := GVL_STATE.G_Window_Sensors[L_i];
    GVL_HMI_SECURITY.G_Window_Bypass[L_i] := GVL_CONFIG.G_Security_Config.bypass_windows[L_i];

    IF GVL_STATE.G_Window_Sensors[L_i] AND NOT GVL_CONFIG.G_Security_Config.bypass_windows[L_i] THEN
        L_Window_Count := L_Window_Count + 1;
    END_IF;
END_FOR;

GVL_HMI_SECURITY.G_Motion_Active_Count := L_Motion_Count;
GVL_HMI_SECURITY.G_Door_Active_Count := L_Door_Count;
GVL_HMI_SECURITY.G_Window_Active_Count := L_Window_Count;
GVL_HMI_SECURITY.G_Total_Active_Count := L_Motion_Count + L_Door_Count + L_Window_Count;

IF GVL_ALARM.G_Security_Alarm THEN
    GVL_HMI_SECURITY.G_Status_Level := 3;
ELSIF GVL_ALARM.G_Security_Armed AND (GVL_HMI_SECURITY.G_Total_Active_Count > 0) THEN
    GVL_HMI_SECURITY.G_Status_Level := 2;
ELSIF GVL_ALARM.G_Security_Armed THEN
    GVL_HMI_SECURITY.G_Status_Level := 1;
ELSE
    GVL_HMI_SECURITY.G_Status_Level := 0;
END_IF;

// >>> BULK_SYNC_ANCHOR: PRG_HMI_Security_Dashboard <<<
END_PROGRAM

(* ---- PRG_HMI_Security_IO_Map_Dashboard.st ---- *)
PROGRAM PRG_HMI_Security_IO_Map_Dashboard
VAR
    L_i : INT;
    L_Map_Index : INT;
    L_Glass_Index : INT;
END_VAR

GVL_HMI_SECURITY_IO_MAP.G_Any_Invalid_Map := FALSE;
GVL_HMI_SECURITY_IO_MAP.G_Group_2F_Active := GVL_IO.DI_Security_2F_Group;

FOR L_i := 1 TO GVL_CONSTANTS.C_MAX_DOOR_SENSORS DO
    L_Map_Index := GVL_CONFIG.G_Door_Map[L_i];
    GVL_HMI_SECURITY_IO_MAP.G_Door_Map[L_i] := L_Map_Index;
    GVL_HMI_SECURITY_IO_MAP.G_Door_Map_Valid[L_i] :=
        (L_Map_Index > 0) AND (L_Map_Index <= GVL_CONSTANTS.C_MAX_SECURITY_SENSORS);

    IF GVL_HMI_SECURITY_IO_MAP.G_Door_Map_Valid[L_i] THEN
        GVL_HMI_SECURITY_IO_MAP.G_Door_Raw_Open[L_i] := GVL_IO.DI_Security_Open[L_Map_Index];
    ELSE
        GVL_HMI_SECURITY_IO_MAP.G_Door_Raw_Open[L_i] := FALSE;
        GVL_HMI_SECURITY_IO_MAP.G_Any_Invalid_Map := TRUE;
    END_IF;
END_FOR;

FOR L_i := 1 TO GVL_CONSTANTS.C_MAX_ZONES DO
    L_Map_Index := GVL_CONFIG.G_Window_Map[L_i];
    GVL_HMI_SECURITY_IO_MAP.G_Window_Map[L_i] := L_Map_Index;
    GVL_HMI_SECURITY_IO_MAP.G_Window_Uses_Open_Input[L_i] := FALSE;
    GVL_HMI_SECURITY_IO_MAP.G_Window_Uses_Glass_Input[L_i] := FALSE;
    GVL_HMI_SECURITY_IO_MAP.G_Window_Overridden_By_2F_Group[L_i] := (L_i = 16);
    GVL_HMI_SECURITY_IO_MAP.G_Window_Raw_Open[L_i] := FALSE;

    IF L_Map_Index > 0 THEN
        IF L_Map_Index <= GVL_CONSTANTS.C_MAX_SECURITY_SENSORS THEN
            GVL_HMI_SECURITY_IO_MAP.G_Window_Map_Valid[L_i] := TRUE;
            GVL_HMI_SECURITY_IO_MAP.G_Window_Uses_Open_Input[L_i] := TRUE;
            GVL_HMI_SECURITY_IO_MAP.G_Window_Raw_Open[L_i] := GVL_IO.DI_Security_Open[L_Map_Index];
        ELSE
            L_Glass_Index := L_Map_Index - GVL_CONSTANTS.C_MAX_SECURITY_SENSORS;
            IF (L_Glass_Index >= 1) AND (L_Glass_Index <= GVL_CONSTANTS.C_MAX_SECURITY_SENSORS) THEN
                GVL_HMI_SECURITY_IO_MAP.G_Window_Map_Valid[L_i] := TRUE;
                GVL_HMI_SECURITY_IO_MAP.G_Window_Uses_Glass_Input[L_i] := TRUE;
                GVL_HMI_SECURITY_IO_MAP.G_Window_Raw_Open[L_i] := GVL_IO.DI_Security_Glass[L_Glass_Index];
            ELSE
                GVL_HMI_SECURITY_IO_MAP.G_Window_Map_Valid[L_i] := FALSE;
                GVL_HMI_SECURITY_IO_MAP.G_Any_Invalid_Map := TRUE;
            END_IF;
        END_IF;
    ELSE
        GVL_HMI_SECURITY_IO_MAP.G_Window_Map_Valid[L_i] := FALSE;
        GVL_HMI_SECURITY_IO_MAP.G_Any_Invalid_Map := TRUE;
    END_IF;
END_FOR;

IF GVL_HMI_SECURITY_IO_MAP.G_Any_Invalid_Map THEN
    GVL_HMI_SECURITY_IO_MAP.G_Status_Text := 'Security IO map has invalid entries';
ELSE
    GVL_HMI_SECURITY_IO_MAP.G_Status_Text := 'Security IO map valid';
END_IF;

// >>> BULK_SYNC_ANCHOR: PRG_HMI_Security_IO_Map_Dashboard <<<
END_PROGRAM

(* ---- PRG_HMI_Water_Dashboard.st ---- *)
PROGRAM PRG_HMI_Water_Dashboard
VAR
    L_i : INT;
    L_Movement_Timeout_MS : UDINT;
END_VAR

L_Movement_Timeout_MS := GVL_CONSTANTS.C_MS_IN_SECOND * 10;

FOR L_i := 1 TO 4 DO
    GVL_HMI.G_HMI_Water_Emergency_Open_Active[L_i] := GVL_WATER_EMERGENCY_OPEN.G_Open_Active[L_i];
    GVL_HMI.G_HMI_Water_Emergency_Open_Remaining_MS[L_i] := GVL_WATER_EMERGENCY_OPEN.G_Open_Remaining_MS[L_i];
    GVL_HMI.G_HMI_Water_Emergency_Open_Count_Today[L_i] := GVL_WATER_EMERGENCY_OPEN.G_Open_Count_Today[L_i];
END_FOR;

GVL_HMI.G_HMI_Water_Emergency_Open_Any_Active := GVL_WATER_EMERGENCY_OPEN.G_Any_Open_Active;
GVL_HMI.G_HMI_Water_Emergency_Open_Last_Accepted := GVL_WATER_EMERGENCY_OPEN.G_Last_Request_Accepted;
GVL_HMI.G_HMI_Water_Emergency_Open_Last_Denied := GVL_WATER_EMERGENCY_OPEN.G_Last_Request_Denied;
GVL_HMI.G_HMI_Water_Emergency_Open_Last_Denial_Code := GVL_WATER_EMERGENCY_OPEN.G_Last_Denial_Code;
GVL_HMI.G_HMI_Water_Emergency_Open_Last_Event_Group := GVL_WATER_EMERGENCY_OPEN.G_Last_Event_Group;
GVL_HMI.G_HMI_Water_Emergency_Open_Last_Event_MS := GVL_WATER_EMERGENCY_OPEN.G_Last_Event_MS;
GVL_HMI.G_HMI_Water_Emergency_Open_Status_Text := GVL_WATER_EMERGENCY_OPEN.G_Status_Text;

IF GVL_WATER_EMERGENCY_OPEN.G_Last_Request_Denied THEN
    GVL_HMI.G_HMI_Water_Emergency_Open_Status_Level := 2;
ELSIF GVL_WATER_EMERGENCY_OPEN.G_Any_Open_Active THEN
    GVL_HMI.G_HMI_Water_Emergency_Open_Status_Level := 1;
ELSE
    GVL_HMI.G_HMI_Water_Emergency_Open_Status_Level := 0;
END_IF;

FOR L_i := 1 TO 6 DO
    GVL_HMI.G_HMI_Water_Valve_Command_Open[L_i] := GVL_WATER_OUTPUT.DO_Water_Local_Valve_Open[L_i];
    GVL_HMI.G_HMI_Water_Valve_Command_Close[L_i] := GVL_WATER_OUTPUT.DO_Water_Local_Valve_Close[L_i];
END_FOR;

GVL_HMI.G_HMI_Water_Valve_Command_Open[7] := GVL_WATER_OUTPUT.DO_Water_Valve_35_Open;
GVL_HMI.G_HMI_Water_Valve_Command_Close[7] := GVL_WATER_OUTPUT.DO_Water_Valve_35_Close;
GVL_HMI.G_HMI_Water_Valve_Command_Open[8] := GVL_WATER_OUTPUT.DO_Water_Valve_36_Open;
GVL_HMI.G_HMI_Water_Valve_Command_Close[8] := GVL_WATER_OUTPUT.DO_Water_Valve_36_Close;

FOR L_i := 1 TO 8 DO
    GVL_HMI.G_HMI_Water_Valve_Open_FB[L_i] := GVL_STATE.G_Water_Zone_Open_FB[L_i];
    GVL_HMI.G_HMI_Water_Valve_Close_FB[L_i] := GVL_STATE.G_Water_Zone_Close_FB[L_i];
    GVL_HMI.G_HMI_Water_Valve_Movement_Timeout_MS[L_i] := L_Movement_Timeout_MS;
    GVL_HMI.G_HMI_Water_Valve_Open_Fault[L_i] := GVL_STATUS.G_Diagnostics.Water_Zone_Open_Fault[L_i];
    GVL_HMI.G_HMI_Water_Valve_Close_Fault[L_i] := GVL_STATUS.G_Diagnostics.Water_Zone_Close_Fault[L_i];
    GVL_HMI.G_HMI_Water_Valve_Critical_Close_Fault[L_i] := GVL_STATUS.G_Diagnostics.Water_Zone_Critical_Close_Fault[L_i];
    GVL_HMI.G_HMI_Water_Valve_Open_Blocked[L_i] := GVL_STATUS.G_Diagnostics.Water_Zone_Open_Blocked[L_i];
END_FOR;

GVL_HMI.G_HMI_Water_Valve_Open_Block_Active := GVL_STATUS.G_Diagnostics.Water_Open_Block_Active;
GVL_HMI.G_HMI_Water_Valve_Open_Block_Text := GVL_STATUS.G_Diagnostics.Water_Open_Block_Text;
GVL_HMI.G_HMI_Water_Valve_Service_Last_Reset_Accepted := GVL_WATER_VALVE_SERVICE.G_Last_Reset_Accepted;
GVL_HMI.G_HMI_Water_Valve_Service_Last_Reset_Denied := GVL_WATER_VALVE_SERVICE.G_Last_Reset_Denied;
GVL_HMI.G_HMI_Water_Valve_Service_Last_Reset_Denial_Code := GVL_WATER_VALVE_SERVICE.G_Last_Reset_Denial_Code;
GVL_HMI.G_HMI_Water_Valve_Service_Last_Reset_Valve_Index := GVL_WATER_VALVE_SERVICE.G_Last_Reset_Valve_Index;
GVL_HMI.G_HMI_Water_Valve_Service_Last_Reset_MS := GVL_WATER_VALVE_SERVICE.G_Last_Reset_MS;
GVL_HMI.G_HMI_Water_Valve_Service_Status_Text := GVL_WATER_VALVE_SERVICE.G_Status_Text;

GVL_HMI.G_HMI_Water_Valve_Close_Fault_Active := GVL_STATUS.G_Diagnostics.Water_Close_Fault_Active;
GVL_HMI.G_HMI_Water_Valve_Main_Shutdown_Recommended := GVL_STATUS.G_Diagnostics.Water_Main_Shutdown_Recommended;
GVL_HMI.G_HMI_Water_Valve_Localization_Failed := GVL_STATUS.G_Diagnostics.Water_Localization_Failed;
GVL_HMI.G_HMI_Water_Valve_Close_Fault_Text := GVL_STATUS.G_Diagnostics.Water_Close_Fault_Text;
GVL_HMI.G_HMI_Water_Valve_Escalation_Text := GVL_STATUS.G_Diagnostics.Water_Escalation_Text;

IF GVL_STATUS.G_Diagnostics.Water_Close_Fault_Active THEN
    GVL_HMI.G_HMI_Water_Valve_Status_Level := 2;
ELSIF GVL_STATUS.G_Diagnostics.Water_Open_Block_Active OR
      GVL_STATUS.G_Diagnostics.Water_Main_Shutdown_Recommended OR
      GVL_STATUS.G_Diagnostics.Water_Localization_Failed THEN
    GVL_HMI.G_HMI_Water_Valve_Status_Level := 1;
ELSE
    GVL_HMI.G_HMI_Water_Valve_Status_Level := 0;
END_IF;

// >>> BULK_SYNC_ANCHOR: PRG_HMI_Water_Dashboard <<<
END_PROGRAM

(* ---- PRG_Input_Processing.st ---- *)
PROGRAM PRG_Input_Processing
VAR
    L_i : INT;
    L_TempDelta : REAL;
    L_HumDelta : REAL;
END_VAR

GVL_INPUT.IN_Last_Update_MS := GVL_TIME_SERVICE.G_Now_MS;
GVL_INPUT.IN_Source_Valid := GVL_STATUS.G_Is_Active_PLC;

GVL_INPUT.IN_Validation_Failed := FALSE;
GVL_INPUT.IN_Anomaly_Detected := FALSE;
GVL_INPUT.IN_Validation_Reason := '';
GVL_INPUT.IN_Anomaly_Reason := '';
GVL_INPUT.IN_Last_Invalid_Zone := 0;

GVL_INPUT.IN_Min_Zone_Confidence := 1.0;
GVL_INPUT.IN_Worst_Zone := 0;

GVL_INPUT.IN_Input_Degraded := GVL_STATUS.G_Diagnostics.Subsystem_Degraded;
GVL_INPUT.IN_Sensor_Fault := GVL_STATUS.G_Diagnostics.Sensor_Fault;

FOR L_i := 1 TO GVL_CONSTANTS.C_MAX_ZONES DO

    GVL_INPUT.IN_Room_Temps[L_i] := GVL_STATE.G_Room_Temps[L_i];
    GVL_INPUT.IN_Room_Hum[L_i] := GVL_STATE.G_Room_Hum[L_i];

    L_TempDelta := ABS(GVL_INPUT.IN_Room_Temps[L_i] - GVL_INPUT.IN_Room_Temp_Prev[L_i]);
    L_HumDelta := ABS(GVL_INPUT.IN_Room_Hum[L_i] - GVL_INPUT.IN_Room_Hum_Prev[L_i]);

    // Default confidence
    GVL_INPUT.IN_Room_Temp_Confidence[L_i] := 1.0;
    GVL_INPUT.IN_Room_Hum_Confidence[L_i] := 1.0;

    // Spike reduces confidence
    IF L_TempDelta > GVL_INPUT_VALIDATION_CONFIG.G_Room_Temp_Spike_Threshold THEN
        GVL_INPUT.IN_Room_Temp_Confidence[L_i] := 0.3;
        GVL_INPUT.IN_Anomaly_Detected := TRUE;
    END_IF;

    IF L_HumDelta > GVL_INPUT_VALIDATION_CONFIG.G_Room_Hum_Spike_Threshold THEN
        GVL_INPUT.IN_Room_Hum_Confidence[L_i] := 0.3;
        GVL_INPUT.IN_Anomaly_Detected := TRUE;
    END_IF;

    // Stuck reduces confidence
    IF L_TempDelta < GVL_INPUT_VALIDATION_CONFIG.G_Room_Temp_Stuck_Epsilon THEN
        IF (GVL_TIME_SERVICE.G_Now_MS - GVL_INPUT.IN_Last_Change_MS[L_i]) > GVL_INPUT_VALIDATION_CONFIG.G_Sensor_Stuck_Timeout_MS THEN
            GVL_INPUT.IN_Room_Temp_Confidence[L_i] := 0.2;
        END_IF;
    ELSE
        GVL_INPUT.IN_Last_Change_MS[L_i] := GVL_TIME_SERVICE.G_Now_MS;
    END_IF;

    // Combined zone confidence
    GVL_INPUT.IN_Zone_Confidence[L_i] :=
        (GVL_INPUT.IN_Room_Temp_Confidence[L_i] + GVL_INPUT.IN_Room_Hum_Confidence[L_i]) / 2.0;

    IF GVL_INPUT.IN_Zone_Confidence[L_i] < GVL_INPUT.IN_Min_Zone_Confidence THEN
        GVL_INPUT.IN_Min_Zone_Confidence := GVL_INPUT.IN_Zone_Confidence[L_i];
        GVL_INPUT.IN_Worst_Zone := L_i;
    END_IF;

    GVL_INPUT.IN_Room_Temp_Prev[L_i] := GVL_INPUT.IN_Room_Temps[L_i];
    GVL_INPUT.IN_Room_Hum_Prev[L_i] := GVL_INPUT.IN_Room_Hum[L_i];

END_FOR;

// >>> BULK_SYNC_ANCHOR: PRG_Input_Processing <<<

(* ---- PRG_IO_Read.st ---- *)
PROGRAM PRG_IO_Read
// ==============================================================================
// IO READ — deterministic physical input acquisition phase map.
// ==============================================================================
// Execution order is preserved from the former monolithic PRG_IO_Read body.
// No gating, shedding or behavior changes are applied here.
// ==============================================================================

PRG_IO_Read_Phase_01_Module_Health();
PRG_IO_Read_Phase_02_Discrete_Debounce();
PRG_IO_Read_Phase_03_Environment_Sensors();
PRG_IO_Read_Phase_04_Heating_Manifold_Sensors();
PRG_IO_Read_Phase_05_Gas_DHW_Water_Feedback();

// >>> BULK_SYNC_ANCHOR: PRG_IO_Read <<<
END_PROGRAM

(* ---- PRG_IO_Read_Discrete_01_Lighting_Sockets.st ---- *)
PROGRAM PRG_IO_Read_Discrete_01_Lighting_Sockets
VAR
    L_i : INT;
    L_Debounce_Time : TIME := T#100MS;

    fbDebounce_Switches : ARRAY[1..GVL_CONSTANTS.C_MAX_LIGHT_ZONES] OF FB_System_Timer;
    fbDebounce_Motion : ARRAY[1..GVL_CONSTANTS.C_MAX_LIGHT_ZONES] OF FB_System_Timer;
END_VAR

FOR L_i := 1 TO GVL_CONSTANTS.C_MAX_LIGHT_ZONES DO
    fbDebounce_Switches[L_i](
        IN := GVL_IO.DI_Lighting_Switches[L_i],
        PT := L_Debounce_Time,
        VI_System_Time_MS := GVL_STATUS.G_System_Time_MS
    );
    GVL_STATE.G_Physical_Switches[L_i] := fbDebounce_Switches[L_i].Q;

    fbDebounce_Motion[L_i](
        IN := GVL_IO.DI_Motion_Sensors[L_i],
        PT := L_Debounce_Time,
        VI_System_Time_MS := GVL_STATUS.G_System_Time_MS
    );
    GVL_STATE.G_Motion_Sensors[L_i] := fbDebounce_Motion[L_i].Q;
END_FOR;

FOR L_i := 1 TO GVL_CONSTANTS.C_MAX_SOCKETS DO
    GVL_STATE.G_Socket_Switches[L_i] := GVL_IO.DI_Socket_Switches[L_i];
END_FOR;

// >>> BULK_SYNC_ANCHOR: PRG_IO_Read_Discrete_01_Lighting_Sockets <<<
END_PROGRAM

(* ---- PRG_IO_Read_Discrete_02_Security_Openings.st ---- *)
PROGRAM PRG_IO_Read_Discrete_02_Security_Openings
VAR
    L_i : INT;
    L_Map_Index : INT;
    L_Glass_Index : INT;
    L_Debounce_Time : TIME := T#100MS;

    fbDebounce_Security_Open : ARRAY[1..GVL_CONSTANTS.C_MAX_SECURITY_SENSORS] OF FB_System_Timer;
    fbDebounce_Security_Glass : ARRAY[1..GVL_CONSTANTS.C_MAX_SECURITY_SENSORS] OF FB_System_Timer;
    fbDebounce_Group_2F : FB_System_Timer;
END_VAR

FOR L_i := 1 TO GVL_CONSTANTS.C_MAX_SECURITY_SENSORS DO
    fbDebounce_Security_Open[L_i](
        IN := GVL_IO.DI_Security_Open[L_i],
        PT := L_Debounce_Time,
        VI_System_Time_MS := GVL_STATUS.G_System_Time_MS
    );

    fbDebounce_Security_Glass[L_i](
        IN := GVL_IO.DI_Security_Glass[L_i],
        PT := L_Debounce_Time,
        VI_System_Time_MS := GVL_STATUS.G_System_Time_MS
    );
END_FOR;

fbDebounce_Group_2F(
    IN := GVL_IO.DI_Security_2F_Group,
    PT := L_Debounce_Time,
    VI_System_Time_MS := GVL_STATUS.G_System_Time_MS
);

FOR L_i := 1 TO GVL_CONSTANTS.C_MAX_DOOR_SENSORS DO
    GVL_STATE.G_Door_Sensors[L_i] := FALSE;
    IF GVL_CONFIG.G_Door_Map[L_i] > 0 AND GVL_CONFIG.G_Door_Map[L_i] <= GVL_CONSTANTS.C_MAX_SECURITY_SENSORS THEN
        GVL_STATE.G_Door_Sensors[L_i] := fbDebounce_Security_Open[GVL_CONFIG.G_Door_Map[L_i]].Q;
    END_IF;
END_FOR;

FOR L_i := 1 TO GVL_CONSTANTS.C_MAX_ZONES DO
    GVL_STATE.G_Window_Sensors[L_i] := FALSE;
    L_Map_Index := GVL_CONFIG.G_Window_Map[L_i];
    IF L_Map_Index > 0 THEN
        IF L_Map_Index <= GVL_CONSTANTS.C_MAX_SECURITY_SENSORS THEN
            GVL_STATE.G_Window_Sensors[L_i] := fbDebounce_Security_Open[L_Map_Index].Q;
        ELSE
            L_Glass_Index := L_Map_Index - GVL_CONSTANTS.C_MAX_SECURITY_SENSORS;
            IF (L_Glass_Index >= 1) AND (L_Glass_Index <= GVL_CONSTANTS.C_MAX_SECURITY_SENSORS) THEN
                GVL_STATE.G_Window_Sensors[L_i] := fbDebounce_Security_Glass[L_Glass_Index].Q;
            END_IF;
        END_IF;
    END_IF;
END_FOR;

GVL_STATE.G_Window_Sensors[16] := fbDebounce_Group_2F.Q;

// >>> BULK_SYNC_ANCHOR: PRG_IO_Read_Discrete_02_Security_Openings <<<
END_PROGRAM

(* ---- PRG_IO_Read_Manifold_02_Temperature_Status.st ---- *)
PROGRAM PRG_IO_Read_Manifold_02_Temperature_Status
VAR
    L_i : INT;

    fbCalib_Manifold_T_Supply : ARRAY[1..GVL_CONSTANTS.C_MAX_MANIFOLDS] OF FB_Sensor_Calibration_Processor;
    fbCalib_Manifold_T_Return : ARRAY[1..GVL_CONSTANTS.C_MAX_MANIFOLDS] OF FB_Sensor_Calibration_Processor;
END_VAR

FOR L_i := 1 TO GVL_CONSTANTS.C_MAX_MANIFOLDS DO
    IF GVL_IO.AI_Manifold_Temps_Supply[L_i].wStatus = 0 THEN
        fbCalib_Manifold_T_Supply[L_i](
            VI_Raw_Value := GVL_IO.AI_Manifold_Temps_Supply[L_i].rValue,
            VI_Record := GVL_CONFIG.G_Calib_Manifold_T_Supply[L_i]
        );
        GVL_STATE.G_Manifold_T_Supply[L_i] := fbCalib_Manifold_T_Supply[L_i].VO_Calibrated_Value;
    END_IF;

    fbCalib_Manifold_T_Return[L_i](
        VI_Raw_Value := INT_TO_REAL(GVL_IO.AI_Manifold_Temps_Return[L_i]) / 10.0,
        VI_Record := GVL_CONFIG.G_Calib_Manifold_T_Return[L_i]
    );
    GVL_STATE.G_Manifold_T_Return[L_i] := fbCalib_Manifold_T_Return[L_i].VO_Calibrated_Value;
    GVL_STATE.G_Manifold_End_Switches[L_i] := GVL_IO.DI_Manifold_End_Switches[L_i];
END_FOR;

// >>> BULK_SYNC_ANCHOR: PRG_IO_Read_Manifold_02_Temperature_Status <<<
END_PROGRAM

(* ---- PRG_IO_Read_Phase_01_Module_Health.st ---- *)
PROGRAM PRG_IO_Read_Phase_01_Module_Health
VAR
    fbIO_Watchdog_1 : FB_IO_Module_Watchdog;
    fbIO_Watchdog_2 : FB_IO_Module_Watchdog;
    fbDiagEventManager : FB_Diagnostics_Event_Manager;
    L_IO_Error_Active : BOOL;
END_VAR

fbIO_Watchdog_1(
    VI_System_Time_MS := GVL_STATUS.G_System_Time_MS,
    VI_Module_ID := 1,
    VI_Heartbeat_Signal := GVL_IO.DI_Module_1_Heartbeat,
    VI_Timeout_MS := 2000
);

fbIO_Watchdog_2(
    VI_System_Time_MS := GVL_STATUS.G_System_Time_MS,
    VI_Module_ID := 2,
    VI_Heartbeat_Signal := GVL_IO.DI_Module_2_Heartbeat,
    VI_Timeout_MS := 2000
);

GVL_STATUS.G_IO_Modules_Online[1] := fbIO_Watchdog_1.VO_Module_Online;
GVL_STATUS.G_IO_Modules_Online[2] := fbIO_Watchdog_2.VO_Module_Online;

L_IO_Error_Active := fbIO_Watchdog_1.VO_Error_Active OR fbIO_Watchdog_2.VO_Error_Active;

fbDiagEventManager(
    VI_Code := 16#E001,
    VI_Severity := 4,
    VI_Active := NOT fbIO_Watchdog_1.VO_Module_Online,
    VI_Timestamp := GVL_STATUS.G_System_Time_MS,
    VI_Source := 1,
    VIO_Events := GVL_STATUS.G_Diagnostics_Events,
    VIO_Count := GVL_STATUS.G_Diagnostics_Count
);

fbDiagEventManager(
    VI_Code := 16#E002,
    VI_Severity := 4,
    VI_Active := NOT fbIO_Watchdog_2.VO_Module_Online,
    VI_Timestamp := GVL_STATUS.G_System_Time_MS,
    VI_Source := 2,
    VIO_Events := GVL_STATUS.G_Diagnostics_Events,
    VIO_Count := GVL_STATUS.G_Diagnostics_Count
);

// >>> BULK_SYNC_ANCHOR: PRG_IO_Read_Phase_01_Module_Health <<<
END_PROGRAM

(* ---- PRG_IO_Read_Phase_02_Discrete_Debounce.st ---- *)
PROGRAM PRG_IO_Read_Phase_02_Discrete_Debounce
// ==============================================================================
// IO READ PHASE 02 — discrete input debounce and mapping.
// ==============================================================================
// Execution order is preserved from the former phase body.
// No gating, shedding or behavior changes are applied here.
// ==============================================================================

PRG_IO_Read_Discrete_01_Lighting_Sockets();
PRG_IO_Read_Discrete_02_Security_Openings();
PRG_IO_Read_Discrete_03_Safety_Sensors();

// >>> BULK_SYNC_ANCHOR: PRG_IO_Read_Phase_02_Discrete_Debounce <<<
END_PROGRAM
